(* CODESYS project ApplicationBase.library
   Author: FS
   Version: 1.0.8
   Description: All sample code provided by Beckhoff Automation LLC are for illustrative purposes only and are provided “as is” and without any warranties, express or implied. Actual implementations in applications will vary significantly. Beckhoff Automation LLC shall have no liability for, and does not waive any rights in relation to, any code samples that it provides or the use of such code samples for any purpose.
   Title: ApplicationBase
   DefaultNamespace: ApplicationBase
   Placeholder: ApplicationBase
   Company: Beckhoff Automation LLC

Project tree, tasks and I/O mapping:
  libraries: Tc2_DataExchange, 3.4.2.0 (Beckhoff Automation GmbH); Tc2_EtherCAT, 3.7.1.0 (Beckhoff Automation GmbH); Tc2_IoFunctions, 3.4.5.0 (Beckhoff Automation GmbH); Tc2_Math, 3.5.1.0 (Beckhoff Automation GmbH); Tc2_MC2, 3.3.72.0 (Beckhoff Automation GmbH); Tc2_MC2_Drive, 3.3.54.0 (Beckhoff Automation GmbH); Tc2_NcKinematicTransformation, 3.2.11.0 (Beckhoff Automation GmbH); Tc2_SerialCom, 3.4.6.0 (Beckhoff Automation GmbH); Tc2_Standard, 3.4.5.0 (Beckhoff Automation GmbH); Tc2_System, 3.10.1.0 (Beckhoff Automation GmbH); Tc2_TcpIp, 3.4.4.0 (Beckhoff Automation GmbH); Tc2_Utilities, 3.10.1.0 (Beckhoff Automation GmbH); Tc3_DynamicMemory, 1.1.4.0 (Beckhoff Automation GmbH); Tc3_EventLogger, 3.3.13.0 (Beckhoff Automation GmbH); Tc3_JsonXml, 3.4.7.0 (Beckhoff Automation GmbH); Tc3_Module, 3.4.5.0 (Beckhoff Automation GmbH); Tc3_PackML_V3, 1.0.6.0 (Beckhoff Automation GmbH)
  _Interface/
    interface I_Base
    interface I_Command: Execute
    interface I_Disposable: Dispose
    interface I_Enablable: Disable, Enable, Enabled
    interface I_Initializable: Initialize, Initialized
    interface I_Override: Override
    interface I_Resettable: Reset
    interface I_Simulatable: Simulated
    interface I_Stoppable: Stop, Stopped
    interface I_TaskResult: Busy, Error, ErrorId
    interface I_ToString: ToString
  _Internal/
    Collection/
      Interface/
        interface I_Collection: AddItem, Clear, Count, IsEmpty, RemoveItem
        interface I_Enumerator: Current, CurrentItem, MoveToNext, ResetIterator
      function block Collection [ST]: FillGaps, AddItem, Clear, Count, Current, CurrentItem, IsEmpty, MoveToNext, RemoveItem, ResetIterator
    CollectionPeeker/
      Interface/
        interface I_CollectionPeeker: CollectionName, FirstItem, LastItem, MoveDownOne, MoveUpOne, PageDown, PageUp, PeekAt, Refresh
        interface I_Peekable: AcceptPeeker
        interface I_Peeker: PeekCollection
      function block CollectionPeeker [ST]: RefreshItems, UpdateEndItem, UpdateFirstItem, CollectionName, FirstItem, Items, LastItem, MoveDownOne, MoveUpOne, PageDown, PageUp, PeekAt, PeekCollection, Refresh
    Component/
      Interface/
        interface I_ComponentCollection: Accept, Count, GetAtIndex, GetComponentByName
        interface I_ContainComponents: Components, DeregisterComponent, DeregisterCyclic, DeregisterInitialize, RegisterComponent, RegisterCyclic, RegisterInitialize
      function block ComponentCollection [ST]: Accept, AddComponent, Count, GetAtIndex, GetComponentByName, RemoveComponent
    Cyclic/
      Interface/
        interface I_Cyclic: CyclicLogic
      function block CyclicRunner [ST]: AddCallee, CallAll, RemoveCallee
    Events/
      function block TcEventClassArguments [ST]: AddString, Clear, Event
    Initialize/
      function block Initializer [ST]: AddInitialize, Initialized, Initializing, RemoveInitialize
    List/
      Interface/
        interface I_List: ContainsItem, GetAtIndex, InsertAtIndex, RemoveAtIndex
      function block List [ST]: AddItem, Clear, RemoveItem, CountListItems, ContainsItem, Count, GetAtIndex, InsertAtIndex, RemoveAtIndex
    Module/
      Interface/
        interface I_ContainModules: DeregisterCyclic, DeregisterInitialize, DeregisterModule, Modules, RegisterCyclic, RegisterInitialize, RegisterModule
        interface I_ModuleCollection: Accept, Count, GetAtIndex, GetModuleByName
      function block ModuleCollection [ST]: Accept, AddModule, Count, GetAtIndex, GetModuleByName, RemoveModule
    MotionTasks/
      AX5000/
        DUT/
          P_0_0074/
            data type ST_IDN_P_0_0074
            data type ST_IDN_P_0_0074_UDINT
          P_0_0074_LREAL/
            data type ST_IDN_P_0_0074_LREAL
          data type ST_AX5000AmpToNm
        function block MotionTask_AX5000AmpToNm [ST]: ActCurrent, ActTorque, Busy, CyclicLogic, Error, ErrorId, Execute
      Base/
        DUT/
          data type ST_TaskState
        function block MotionTask [ST]: Axis, Busy, CyclicLogic, Error, ErrorId, Execute, Name
        function block MotionTaskCollection [ST]: Busy, Error, ErrorId, ErrorTask, AddTask, CyclicLogic, FB_Init, RemoveTaskByInstance, Reset
      Coupling/
        function block MotionCoupleTask_Gearing [ST]: BufferMode, Busy, CyclicLogic, Error, ErrorId, Execute, GearIn, GearInMultiMasterOptions, GearRatioMaster1, GearRatioMaster2, GearRatioMaster3, GearRatioMaster4, Master1, Master2, Master3, Master4
      Home/
        function block MotionHomeTask_CoESetEncoderOffset [ST]: Busy, CyclicLogic, Error, ErrorId, Execute, HomePosition
        function block MotionHomeTask_SetPosition [ST]: Busy, CyclicLogic, Error, ErrorId, Execute, HomePosition
        function block MotionHomeTask_SetPositionOffset [ST]: Busy, CyclicLogic, Error, ErrorId, Execute, Feedback, HomePosition, Memory
        function block MotionHomeTask_SetZeroHere [ST]: Busy, CyclicLogic, Error, ErrorId, Execute
      Interface/
        interface I_AxisRef: Axis
        interface I_MotionJogTask: JogBackwards, JogForward, Mode, Position
        interface I_MotionPowerTask
        interface I_MotionTask: Axis, Name
        interface I_MotionTaskCollection: AddTask, ErrorTask, RemoveTaskByInstance
      Move/
        function block MoveAbsoluteTask [ST]: BufferMode, Busy, CyclicLogic, Error, ErrorId, Execute, MoveOptions, TargetPosition
        function block MoveJogTask [ST]: Busy, CyclicLogic, Error, ErrorId, Execute, JogBackwards, JogForward, Mode, Position
        function block MoveModuloTask [ST]: BufferMode, Busy, CyclicLogic, Direction, Error, ErrorId, Execute, MoveOptions, TargetPosition
        function block MoveRelativeTask [ST]: BufferMode, Busy, CyclicLogic, Error, ErrorId, Execute, MoveOptions, TargetDistance
        function block MoveVelocityTask [ST]: BufferMode, Busy, CyclicLogic, Error, ErrorId, Execute, MoveOptions, TargetVelocity
      Power/
        function block PowerTask [ST]: Busy, CyclicLogic, Disable, Enable, Enabled, Error, ErrorId, Execute, InhibitFeedBackward, InhibitFeedForward, Override
        function block StopTask [ST]: BufferMode, Busy, CyclicLogic, Error, ErrorId, Execute, MoveOptions
      Reset/
        function block CoEExtendedResetTask [ST]: Busy, CyclicLogic, Error, ErrorId, Execute
        function block CoEResetTask [ST]: Busy, CyclicLogic, Error, ErrorId, Execute
        function block SoEResetTask [ST]: Busy, CyclicLogic, Error, ErrorId, Execute
    Null/
      function block NullComponent [ST]
      function block NullItem [ST]
      function block NullModule [ST]: Accept, Components, DeregisterComponent, DeregisterCyclic, DeregisterInitialize, DeregisterModule, DeregisterWithParent, FB_Init, Modules, Name, RegisterComponent, RegisterCyclic, RegisterInitialize, RegisterModule, RegisterWithParent, ResetComponents, ResetModules
    Statemachine/
      Interface/
        interface I_StateList: AddStateAtIndex, GetStateAtIndex, NumberOfStates
      function block StateList [ST]: AddStateAtIndex, GetStateAtIndex, NumberOfStates
    Tracing/
      Interface/
        interface I_ContainTraceArgument: Arguments
        interface I_ContainTracePublisher: Publisher
        interface I_TraceArgument
        interface I_TraceInstanceLogger: LogMessageInstance
        interface I_TraceLogger: LogMessage
        interface I_TraceMessageInfo: Message, MessageId, Severity
        interface I_TracePublisher: Subscribe, Unsubscribe
        interface I_TraceSourceInfo: SourceId, SourceName, TimeStamp
      function block AdsLogger [ST]: FB_Init, LogMessage
      function block LocalLogger [ST]: ClearLog, LogMessage, Messages
      function block TcEventLogger [ST]: FB_Init, LogMessage
      function block TraceMessageInfo [ST]: Message, MessageId, Severity
      function block TraceSourceInfo [ST]: SourceId, SourceName, TimeStamp
      function USINT_To_TcEventSeverity [ST]
    Types/
      data type RegistrationResult
  Component/
    Interface/
      interface I_Component: Accept, DeregisterWithParent, Name, RegisterWithParent
      interface I_ComponentVisitor: VisitComponent
    function block Component [ST]: Accept, DeregisterWithParent, Name, RegisterWithParent, FB_Init
    function block CyclicComponent [ST]: CyclicLogic, DeregisterWithParent, RegisterWithParent
  Components/
    ADS/
      Interface/
        interface I_AdsAccess: AdsRW
        interface I_AdsRW: AmsNetId, AmsPort, Read, ReadBySymbol, Write, WriteBySymbol
      function block AdsReadWrite [ST]: Busy, Error, ErrorId, AdsComMode, AmsNetId, AmsPort, CyclicLogic, Read, ReadBySymbol, Write, WriteBySymbol
    Analog/
      DUT/
        data type ST_AnalogInputStatus_EL30xx
        data type ST_AnalogInputStatus_Generic
      Interface/
        interface I_AnalogChannel_Generic: DataValid, Error, Overrange, Underrange
        interface I_AnalogChannel_Standard: Limit1High, Limit1Low, Limit2High, Limit2Low
        interface I_AnalogInput: RawValue, Value
        interface I_AnalogOutput: RawValue, Value
      function block AnalogInput [ST]: CalibrateCustom, CalibrateLinear, FB_Init, Force, ForceValue, RawValue, Scale, Value
      function block AnalogInput_Generic [ST]: DataValid, Error, FB_Init, Overrange, Underrange
      function block AnalogInput_Standard [ST]: DataValid, Error, FB_Init, Limit1High, Limit1Low, Limit2High, Limit2Low, Overrange, Underrange
      function block AnalogOutput [ST]: CalibrateCustom, CalibrateLinear, FB_Init, Force, ForceValue, RawValue, Scale, Value
    CoE/
      DUT/
        data type ST_TerminalProductInfo
      Interface/
        interface I_CoeAccess: CoE
        interface I_CoeDevice: AdsAddr, Read, Write
      function block CoeDevice [ST]: Busy, Error, ErrorId, AdsAddr, CyclicLogic, Read, Write
      function block NullCoeDevice [ST]: AdsAddr, Busy, CyclicLogic, Error, ErrorId, Read, Write
    Cylinder/
      DUT/
        data type E_CylinderErrorId
        data type E_CylinderState
        data type ST_Cylinder_HMI
      Interface/
        interface I_Cylinder: ExtendTimeout, RetractTimeout
        interface I_CylinderCommand: Extend, Retract
        interface I_CylinderStatus: Extended, Extending, Retracted, Retracting
      function block Cylinder [ST]: CyclicLogic, Busy, Error, ErrorId, Extend, Extended, Extending, ExtendTimeout, Retract, Retracted, Retracting, RetractTimeout, Reset, FB_Init
      function block Cylinder_HMI [ST]: ExtendPermissive, RetractPermissive, ControlObject, CyclicLogic, ExtendCommandName, ExtendedName, FB_Init, RetractCommandName, RetractedName
      function block Cylinder_TcEvents [ST]: GetHighestActiveEventReaction, GetHighestActiveEventSeverity, Reset, SetEventReactions, CyclicLogic, FB_Init
    Digital/
      DUT/
        data type ST_DigitalInput_HMI
        data type ST_DigitalOutput_HMI
      Interface/
        interface I_DigitalInput: IsActive
        interface I_DigitalOutput: On
      Visitor/
        function block ForceVisitor [ST]: Force, VisitComponent
        function block ReleaseAllForceVisitor [ST]: ReleaseForces, VisitComponent, VisitModule
      function block DigitalInput_Combiner [ST]: AddInput, Force, IsActive
      function block DigitalInput_DebounceFallingEdge [ST]: CyclicLogic, DebounceTime, FB_Init, Force, IsActive
      function block DigitalInput_DebounceRisingEdge [ST]: CyclicLogic, DebounceTime, FB_Init, Force, IsActive
      function block DigitalInput_HMI [ST]: ControlObject, CyclicLogic, FB_Init
      function block DigitalInput_NC [ST]: FB_Init, Force, IsActive
      function block DigitalInput_NO [ST]: FB_Init, Force, IsActive
      function block DigitalOutput [ST]: FB_Init, Force, On
      function block DigitalOutput_HMI [ST]: ControlObject, CyclicLogic, FB_Init
    EtherCat/
      DUT/
        global variables EtherCatParameter
        data type ST_EtherCatMasterInfo
        data type ST_EtherCatSyncUnitTaskInfo
      Interface/
        interface I_EcIoDevice: Bootstrap, Configuration, DeviceError, Disabled, Init, InitCmdError, InvalidVPRS, OP, PreOp, SafeOp, State
        interface I_EtherCatDiagnosticEventProvider: RaiseEtherCatDiagnosticEvent, RaiseSyncUnitEvent
        interface I_EtherCatMasterDiagnostic: ConfiguredSlaveCount, GetIoDeviceByAddr, GetIoDeviceByName, LocalAmsNetId, MasterAmsNetId, RegisterEventProvider, SlaveCount
        interface I_IoDevice: IoDataValid
        interface I_SyncUnitTask: IoDataValid, IsHotConnect, SlaveCount
      function block EtherCatIoDevice [ST]: Bootstrap, CoE, Configuration, DeviceError, Disabled, Init, InitCmdError, InvalidVPRS, IoDataValid, OP, PreOp, SafeOp, State, AmsNetId, CyclicLogic, SyncUnit
      function block EtherCatMaster [ST]: FramesWcStatesOk, LookupMasterState, LookupSlaveState, MasterState, SlaveState, ConfiguredSlaveCount, GetIoDeviceByAddr, GetIoDeviceByName, LocalAmsNetId, MasterAmsNetId, RegisterEventProvider, SlaveCount, Initialize, Initialized, Reset, Busy, Error, ErrorId, CyclicLogic, FB_Init, Simulated
      function block EtherCatMaster_TcEvents [ST]: GetHighestActiveEventReaction, GetHighestActiveEventSeverity, RaiseEtherCatDiagnosticEvent, RaiseSyncUnitEvent, Reset, SetEventReactions, FB_Init
      function block SyncUnitTask [ST]: Initialize, Initialized, IoDataValid, IsHotConnect, IsTerminalPartOfSyncUnit, SlaveCount, Busy, Error, ErrorId, CyclicLogic, EventProvider, FB_Init, Simulated
    Recipe/
      Interface/
        interface I_RecipeManagment: AutoLoadChangesToActive, ChangesPending, LoadChangesToActive
      function block RecipeManagment [ST]: CyclicLogic, CompareData, AutoLoadChangesToActive, ChangesPending, LoadChangesToActive, FB_Init
    Safety/
      DUT/
        data type E_SafetyConnection_State
        data type E_SafetyEdm_State
        data type E_SafetyEStop_State
        data type E_SafetyGroup_Diag
        data type E_SafetyGroup_State
        data type E_SafetyMon_State
        data type E_SafetyOrAnd_State
        data type ST_SafetyAddressInfo
        data type ST_SafetyDeviceInfo
        data type ST_SafetyStateDiag
      Interface/
        interface I_InSafetyGroup: SafetyGroup
        interface I_SafetyBase: OK, ResetFunction
        interface I_SafetyModule: AddSafetyComponent, OK, SafetyPlcCoE
        interface I_SafetyReset: Execute, PulseDuration
        interface I_SafetySimulation: SimulateSafetyDiag, SimulateSafetyState
      Reset Function/
        function block SafetyResetPulse [ST]: CyclicLogic, Busy, Error, ErrorId, Execute, PulseDuration
      Visitor/
        function block SafetyOkVisitor [ST]: Check, OK, VisitComponent
        function block SetSafetySimulationVisitor [ST]: Diag, Simulated, State, VisitComponent
      function block SafetyAndOrFB [ST]: CyclicLogic
      function block SafetyBase [ST]: CyclicLogic, OK, Reset, ResetFunction, Simulated, SimulateSafetyDiag, SimulateSafetyState, Busy, Error, ErrorId
      function block SafetyConnectionFB_TcEvents [ST]: CyclicLogic, GetHighestActiveEventReaction, GetHighestActiveEventSeverity, Reset, SetEventReactions, FB_Init
      function block SafetyEdmFB_TcEvents [ST]: CyclicLogic, GetHighestActiveEventReaction, GetHighestActiveEventSeverity, Reset, SetEventReactions, FB_Init, SafetyGroup
      function block SafetyEstopFB_TcEvents [ST]: CyclicLogic, GetHighestActiveEventReaction, GetHighestActiveEventSeverity, Reset, SetEventReactions, ActiveName, FB_Init, SafetyGroup
      function block SafetyGroup_TcEvents [ST]: CyclicLogic, GetHighestActiveEventReaction, GetHighestActiveEventSeverity, Reset, SetEventReactions, AutoResetFaults, FB_Init
      function block SafetyModule [ST]: OnCyclicCall, Initializing, Simulated, SimulateSafetyDiag, SimulateSafetyState, Busy, Error, ErrorId, AddSafetyComponent, FB_Init, OK, Reset, SafetyAddressInfo, SafetyPlcCoE
      function block SafetyMonFB_TcEvents [ST]: CyclicLogic, GetHighestActiveEventReaction, GetHighestActiveEventSeverity, Reset, SetEventReactions, ActiveAlarm, ActiveName, FB_Init, SafetyGroup
    Serial/
      Interface/
        interface I_SerialByteConnection: ByteData, ByteDataRecieved, SendAByte
        interface I_SerialLineControl: rxBuffer, txBuffer
        interface I_SerialStringConnection: SendAString, StringData, StringRecieved
      function block SerialByteConnection [ST]: ByteData, ByteDataRecieved, CyclicLogic, FB_Init, Reset, SendAByte, SetDependencies
      function block SerialLineControl_ADS [ST]: CyclicLogic, rxBuffer, SetConnectionConfig, txBuffer
      function block SerialLineControl_Terminal [ST]: CyclicLogic, FB_Init, rxBuffer, SetConnectionConfig, SetDependencies, txBuffer
      function block SerialStringConnection [ST]: CyclicLogic, FB_Init, Reset, SendAString, SetDependencies, SetSerialConfiguration, StringData, StringRecieved
    Tcp Ip/
      DUT/
        data type ST_TcpIpPayload
      Interface/
        interface I_TcpIpConnection: ConnectionState, IP, Port, RegisterCommand, SendCommand, SendPriorityCommand, Socket
        interface I_TcpIpSubscription: UpdateCommandResult
      function block TcpIpCommandResultFilter [ST]: CyclicLogic, FB_Init, UpdateCommandResult
      function block TcpIpConnection [ST]: CyclicLogic, Initialize, Initialized, EvaluateResponse, GetNextCommand, GetNextPriorityCommand, SendReceiveSequence, ConnectionState, IP, PollTime, Port, ReceiveTimeout, ReconnectionTime, RegisterCommand, SendCommand, SendInterval, SendPriorityCommand, Socket
      global variables TcpIpConnectionParameter
  Events/
    Interface/
      interface I_EventArguments: AddString, Clear
      interface I_EventClass: Arguments, ClearEventById, IsResettable, RaiseEvent, ResetBySeverity, SetEvent
      interface I_EventClassTcEvents: GenerateTcEvents, GetHighestActiveEventSeverity
      interface I_EventReaction: GetHighestActiveEventReaction, SetEventReactions
      interface I_EventReactionTcEvents: GetHighestActiveEventSeverity
    function block TcEventClass [ST]: Dispose, FB_Exit, ClearEventById, GetHighestActiveEventReaction, GetHighestActiveEventSeverity, IsResettable, RaiseEvent, ResetBySeverity, SetEvent, SetEventReactions, CheckEventId, FindActiveSeverity, GetEventAutoResetInstance, GetEventInstance, GetEventTriggerInstance, SetEventTriggerInstance, Reset, Arguments, CyclicLogic, GenerateTcEvents
  HMI/
    DUT/
      data type ST_HmiFunction
    Interface/
      interface I_Button: Active, Name, Permissive
      interface I_HmiFunction: ControlType, Disable, Enable, Enabled, InstancePath, LinkObject
      interface I_Permissive: OK, Set
      interface I_StringCollection: AddString, Clear, Entries
    function block Button [ST]: Active, Name, Permissive
    function block HmiFunction [ST]: ControlObject, ControlType, CyclicLogic, Disable, Enable, Enabled, InstancePath, LinkObject
  Kinematic Group/
    Interface/
      interface I_KinematicGroup: AddAcsAxis, AddMcsAxis, BuildGroup, DissolveGroup, Status
    function block KinematicGroup [ST]: DeregisterWithParent, RegisterWithParent, CyclicLogic, Initialize, Initialized, AddAcsAxis, AddMcsAxis, BuildGroup, DissolveGroup, Override, Status, Reset, Busy, Error, ErrorId
    function block KinematicGroup_TcEvents [ST]: GetHighestActiveEventReaction, GetHighestActiveEventSeverity, Reset, SetEventReactions, CyclicLogic, FB_Init
  Modes/
    Interface/
      interface I_Mode: ChangeMode, CurrentMode
    function block ModeControl [ST]: ChangeMode, CurrentMode
    function block PackMLModeControl [ST]: ChangeMode, CurrentMode, CyclicLogic, StateMachine
  Module/
    Interface/
      interface I_Module: Accept, DeregisterWithParent, Name, RegisterWithParent, ResetComponents, ResetModules
      interface I_ModuleVisitor: VisitModule
    function block Module [ST]: FB_Init, CyclicLogic, OnCyclicCall, DeregisterComponent, DeregisterCyclic, DeregisterInitialize, DeregisterModule, DeregisterWithParent, Initialize, Initialized, Initializing, RegisterComponent, RegisterCyclic, RegisterInitialize, RegisterModule, RegisterWithParent, ResetComponents, ResetModules, Accept, Components, Modules, Name
  Module PackML/
    function block PackMLModule [ST]: FB_Init, Aborted, Aborting, Clearing, Completed, Completing, Execute, Held, Holding, Idle, Resetting, Starting, Stopped, Stopping, Suspended, Suspending, Unholding, Unsuspending, CyclicLogic, Statemachine, StateSelect
  Motion/
    DUT/
      data type ST_AxisPTP_HMI
      data type ST_MotionDefaults
    Interface/
      interface I_Axis: ErrorId, MotionTasks
      interface I_Axis_PTP
      interface I_AxisDynamics: Acceleration, BufferMode, Deceleration, Jerk, MoveOptions, Velocity
      interface I_AxisEnable: InhibitFeedBackward, InhibitFeedForward
      interface I_AxisGear: GearIn, GearInMultiMasterOptions, GearOut, GearRatioMaster1, GearRatioMaster2, GearRatioMaster3, GearRatioMaster4, Master1, Master2, Master3, Master4
      interface I_AxisHome: Home
      interface I_AxisJog: Jog
      interface I_AxisMoveAbsolute: MoveAbsolute
      interface I_AxisMoveModulo: MoveModulo
      interface I_AxisMoveRelative: MoveRelative
      interface I_AxisMoveVelocity: MoveVelocity
      interface I_AxisStatus: ActualAcceleration, ActualPosition, ActualPositionModulo, ActualTorque, ActualVelocity, AxisParameterSet, Enabled, PositionLag, SetAcceleration, SetPosition, SetPositionModulo, SetVelocity, Stopped
      interface I_SlaveAxis
    function block Axis [ST]: FB_Init, RegisterWithParent, CyclicLogic, Acceleration, BufferMode, Deceleration, Jerk, MoveOptions, Velocity, Disable, Enable, Enabled, InhibitFeedBackward, InhibitFeedForward, Override, Home, HomeTask, Initialize, Initialized, Jog, Reset, ResetTask, ActualAcceleration, ActualPosition, ActualPositionModulo, ActualTorque, ActualVelocity, AxisParameterSet, Busy, Error, ErrorId, PositionLag, SetAcceleration, SetPosition, SetPositionModulo, SetVelocity, Stop, Stopped, StopTask, Axis, MotionTasks
    function block Axis_TcEvents [ST]: GetHighestActiveEventReaction, GetHighestActiveEventSeverity, Reset, SetEventReactions, CyclicLogic, FB_Init
    function block AxisPTP [ST]: FB_Init, MoveAbsolute, MoveModulo, MoveRelative, MoveVelocity
    function block AxisPTP_HMI [ST]: DisablePermissive, EnablePermissive, HomePermissive, JogBackwardFastPermissive, JogBackwardSlowPermissive, JogForwardFastPermissive, JogForwardSlowPermissive, MoveAbsolutePermissive, MoveModuloPermissive, MoveRelativePermissive, MoveVelocityPermissive, ResetPermissive, StopPermissive, ControlObject, CyclicLogic, FB_Init
    function block SlaveAxisPTP [ST]: FB_Init, GearIn, GearInMultiMasterOptions, GearOut, GearRatioMaster1, GearRatioMaster2, GearRatioMaster3, GearRatioMaster4, Master1, Master2, Master3, Master4
  Permissive Interlock/
    function block PermissiveInterlock [ST]: Check, OK, Set
  Project Information/
    function F_GetCompany [ST]
    function F_GetTitle [ST]
    function F_GetVersion [ST]
  Statemachine/
    DUT/
      data type ST_PackMLStatemachine_HMI
      data type ST_Statemachine_HMI
    Generic/
      function NextMinorStep [ST]
      function NextStep [ST]
      function SetStep [ST]
      function block State [ST]: Executing, FB_Init, Inactive
      function block Statemachine [ST]: Mode, ChangeState, CurrentState, States, CyclicLogic
      function block Statemachine_HMI [ST]: ControlObject, CyclicLogic, FB_Init
    Interface/
      interface I_ContainStatemachine: Statemachine
      interface I_State: Executing, Inactive
      interface I_Statemachine: ChangeState, CurrentState, Mode, States
    PackML/
      function block NextAvailablePackMLCommands [ST]: GetCommands
      function block PackMLStatemachine [ST]: Mode, CallState, ChangeState, CurrentState, States, CyclicLogic
      function block PackMLStatemachine_HMI [ST]: ControlObject, CyclicLogic, FB_Init
      function block PackMLStatemachine_ModuleIntegrated [ST]: Mode, ChangeState, CurrentState, CyclicLogic, StateComplete, States
  Tracing/
    DUT/
      data type TcEventSeverityExt
    Interface/
      interface I_Trace: Critical, Error, Info, Verbose, Warning
    global variables CoreTrace
    function block Trace [ST]: Critical, Error, Info, LogMessage, Subscribe, TraceLevel, Unsubscribe, Verbose, Warning
  Utilities/
    AnyBuffer/
      DUT/
        data type ST_BufferConfiguration
        data type ST_BufferMetadata
      Interface/
        interface I_AnyBuffer: Clear, Configuration, DeleteAtIndex, isEmpty, isFull, Metadata, PeekAtIndex, PopAtIndex, PopLeft, PopRight, PushAtIndex, PushLeft, PushRight, ReplaceAtIndex
        interface I_AnyBufferStrategy: Clear, isEmpty, isFull
      TypedBuffers/
        function block FifoBuffer [ST]: Clear, FB_Init, isEmpty, isFull, Pop, Push
        function block LifoBuffer [ST]: Clear, FB_Init, isEmpty, isFull, Pop, Push
        function block ListBuffer [ST]: Clear, FB_Init, isEmpty, isFull, Pop, Push, removeOldest
        function block RingBuffer [ST]: AdvanceHead, AdvanceTail, Clear, FB_Init, isEmpty, isFull, Pop, Push
      function block AnyBuffer [ST]: buffer, Clear, Configuration, CountDecrement, CountIncrement, DeleteAtIndex, FB_Exit, FB_Init, FB_Reinit, isEmpty, isFull, Metadata, PeekAtIndex, PopAtIndex, PopLeft, PopRight, PushAtIndex, PushLeft, PushRight, ReplaceAtIndex
    File/
      DUT/
        data type ST_File_HMI
      Interface/
        interface I_FileHandler: ClearDocument, Datatype, LoadFile, nData, Path, pData, ReadSymbol, SaveFile, SymbolName, Timeout, UpdateSymbol
      function block File_HMI [ST]: LoadPermissive, SavePermissive, ControlObject, CyclicLogic, FB_Init
      function block JsonFile [ST]: CyclicLogic, ClearDocument, Datatype, LoadFile, nData, Path, pData, ReadSymbol, SaveFile, SymbolName, Timeout, UpdateSymbol, LoadFileSequence, SaveFileSequence, Reset, Busy, Error, ErrorId
      function block StringHelper [ST]: GetExtensionOrVarName, GetFileNameFromPath, GetFilePath, GetName, GetPath, GetSymbolPath, RemoveFirstChar, RemoveLastChar, StringToCharArray, ValidInput
    Flash/
      function block SyncedSquareWaves [ST]: Initialize, Initialized, CyclicLogic, Wave_0_5Hz, Wave_100Hz, Wave_1Hz, Wave_2Hz, Wave_500Hz, Wave_50Hz, Wave_5Hz
    Force/
      DUT/
        data type E_ForceState
      Interface/
        interface I_ForcibleBool: Force
        interface I_ForcibleInt: Force, ForceValue
      function block ForcibleBool [ST]: ResolveOutput, CurrentForceState, FB_Init, Input, Output, SetForceState
      function block ForcibleInt [ST]: ResolveOutput, CurrentForceState, FB_Init, ForceValue, Input, Output, SetForceState
    Functions/
      function CompareLREAL [ST]
      function CompareModulo [ST]
      function PercentToAnalog [ST]
    Scaling/
      Interface/
        interface I_AnalogScalable: Scale
        interface I_AnalogScale: InputMaximum, InputMinimum, OutputMaximum, OutputMinimum
        interface I_CalibratableLinear: CalibrateLinear
        interface I_CalibrateLinear: Gain, Offset
        interface I_TransformLRealValue: Transform
      function block AnalogScale [ST]: InputMaximum, InputMinimum, OutputMaximum, OutputMinimum, Transform
      function block Calibrate [ST]: Gain, Offset, Transform
    Timing/
      function block Stopwatch [ST]: Elapsed, Lap, Running, Start, Stop
  Version/
    global variables Global_Version
  Visitors/
    Enable/
      function block CheckComponentsEnabledVisitor [ST]: Check, Enabled, VisitComponent
      function block DisableAllComponentsVisitor [ST]: Disable, Enabled, VisitComponent
      function block EnableAllComponentsVisitor [ST]: Enable, Enabled, VisitComponent
    Events/
      function block GetActiveEventSeverityVisitor [ST]: ActiveEventSeverity, FB_Init, VisitComponent, VisitModule
    HMI/
      function block GetSystemTreeJsonHmiVisitor [ST]: Clear, FB_Init, GetTree, VisitComponent, VisitModule
      function block HmiEnableDisableAllVisitor [ST]: DisableHmi, EnableHmi, VisitComponent, VisitModule
    Override/
      function block SetAllOverrideVisitor [ST]: Set, VisitComponent, VisitModule
    PackML Statemachine/
      function block ChangePackMLStateOnAllSubModulesVisitor [ST]: ChangeState, VisitModule
      function block EventReactorPackMLVisitor [ST]: CyclicLogic, FB_Init, VisitComponent, VisitModule
    Reset/
      function block GetComponentsTaskResultVisitor [ST]: Busy, Error, ErrorId, Update, VisitComponent
      function block ResetAllVisitor [ST]: Busy, Error, ErrorId, Reset, VisitComponent, VisitModule
      function block ResetComponentsVisitor [ST]: Busy, Error, ErrorId, Reset, VisitComponent
      function block ResetModulesVisitor [ST]: Busy, Error, ErrorId, Reset, VisitModule
    Statemachine/
      function block ChangeModeOnAllSubModulesVisitor [ST]: ChangeMode, VisitModule
      function block ChangeStateOnAllSubModulesVisitor [ST]: ChangeState, VisitModule
      function block EventReactorVisitor [ST]: CyclicLogic, FB_Init, VisitComponent, VisitModule
    Stop/
      function block StopAllComponentsVisitor [ST]: Stop, Stopped, VisitComponent
  global variables ApplicationBaseMotionParameterNc2
  global variables ApplicationBaseParameter
*)

// _Internal/MotionTasks/AX5000/DUT/P_0_0074/ST_IDN_P_0_0074
TYPE ST_IDN_P_0_0074 :
	STRUCT
		Iq : ARRAY[0..9] OF UDINT; // Amps ( units := A x 100 )
		M  : ARRAY[0..9] OF UDINT; // Newton Meters ( units := Nm x 100 )
	END_STRUCT
END_TYPE

// _Internal/MotionTasks/AX5000/DUT/P_0_0074/ST_IDN_P_0_0074_UDINT
TYPE ST_IDN_P_0_0074_UDINT :
	STRUCT
		Actual	 : UINT;
		_Max	 : UINT;
		Elements : ST_IDN_P_0_0074;
	END_STRUCT
END_TYPE

// _Internal/MotionTasks/AX5000/DUT/P_0_0074_LREAL/ST_IDN_P_0_0074_LREAL
TYPE ST_IDN_P_0_0074_LREAL :
	STRUCT
		Iq : ARRAY[0..9] OF LREAL;
		M  : ARRAY[0..9] OF LREAL;
	END_STRUCT
END_TYPE

// _Internal/MotionTasks/AX5000/DUT/ST_AX5000AmpToNm
TYPE ST_AX5000AmpToNm :
	STRUCT
		Curve	   : ST_IDN_P_0_0074_LREAL; // Contents read in from P-0-0074   ( scaled )
		ActCurrent : LREAL;					// Actual current in Amps           ( units := A )
		ActTorque  : LREAL;					// Actual torque in Newton Meters   ( units := Nm )
	END_STRUCT
END_TYPE

// _Internal/MotionTasks/Base/DUT/ST_TaskState
TYPE ST_TaskState :
	STRUCT
		Name	: T_MaxString;
		Busy	: BOOL;
		Error	: BOOL;
		ErrorId : UDINT;
	END_STRUCT
END_TYPE

// _Internal/Types/RegistrationResult
{attribute 'qualified_only'}
{attribute 'strict'}
{attribute 'to_string'}
TYPE RegistrationResult :
(
	Succeeded := 0,
	NullReference := -1,
	TooManyComponents := -2,
	AlreadyAdded := -3,
	CollectionEmpty := -4,
	NotFoundInCollection := -5
);
END_TYPE

// Components/Analog/DUT/ST_AnalogInputStatus_EL30xx
{attribute 'pack_mode' := '1'}
TYPE ST_AnalogInputStatus_EL30xx :
	STRUCT
		Underrrange : BIT;
		Overrange	: BIT;
		Limit1L		: BIT;
		Limit1H		: BIT;
		Limit2L		: BIT;
		Limit2H		: BIT;
		Error		: BIT;
		TxPDOState	: BIT;
		TxPDOToggle : BIT;
	END_STRUCT
END_TYPE

// Components/Analog/DUT/ST_AnalogInputStatus_Generic
{attribute 'pack_mode' := '1'}
TYPE ST_AnalogInputStatus_Generic :
	STRUCT
		Underrrange : BIT;
		Overrange	: BIT;
		Error		: BIT;
		WcState		: BIT;
	END_STRUCT
END_TYPE

// Components/CoE/DUT/ST_TerminalProductInfo
{attribute 'pack_mode' := '2'}
TYPE ST_TerminalProductInfo : // Parameter 16#1018:0
	STRUCT
		Identity	 : WORD;
		VendorId	 : DINT;
		ProductCode	 : DINT;
		Revision	 : DINT;
		SerialNumber : DINT;
	END_STRUCT
END_TYPE

// Components/Cylinder/DUT/E_CylinderErrorId
{attribute 'qualified_only'}
TYPE E_CylinderErrorId : (
		NoError				  := 0,
		ExtendTimeout		  := 1,
		RetractTimeout		  := 2,
		ExtendedPlausibility  := 3,
		RetractedPlausibility := 4,
		BothSensorsActive	  := 5
	) UDINT;
END_TYPE

// Components/Cylinder/DUT/E_CylinderState
{attribute 'qualified_only'}
TYPE E_CylinderState : (
		Undefined  := 0,
		Extending  := 1,
		Extended   := 2,
		Retracting := 3,
		Retracted  := 4
	);
END_TYPE

// Components/Cylinder/DUT/ST_Cylinder_HMI
TYPE ST_Cylinder_HMI EXTENDS ST_HmiFunction :
	STRUCT
		Busy		  : BOOL;
		Error		  : BOOL;
		ErrorId		  : UDINT;
		Extended	  : BOOL;
		ExtendedName  : STRING := 'Extended';
		Retracted	  : BOOL;
		RetractedName : STRING := 'Retracted';
		Extend		  : Button;
		Retract		  : Button;
	END_STRUCT
END_TYPE

// Components/Digital/DUT/ST_DigitalInput_HMI
TYPE ST_DigitalInput_HMI EXTENDS ST_HmiFunction :
	STRUCT
		Active : BOOL;
		Force  : E_ForceState;
	END_STRUCT
END_TYPE

// Components/Digital/DUT/ST_DigitalOutput_HMI
TYPE ST_DigitalOutput_HMI EXTENDS ST_HmiFunction :
	STRUCT
		On	  : BOOL;
		Force : E_ForceState;
	END_STRUCT
END_TYPE

// Components/EtherCat/DUT/ST_EtherCatMasterInfo
TYPE ST_EtherCatMasterInfo :
	STRUCT
		AmsNetID	  : AMSNETID;
		DevID		  : UINT;
		DevState	  : UINT;
		ChangeCount	  : UINT;
		SlaveCount	  : UINT;
		CfgSlaveCount : UINT;
	END_STRUCT
END_TYPE

// Components/EtherCat/DUT/ST_EtherCatSyncUnitTaskInfo
TYPE ST_EtherCatSyncUnitTaskInfo :
	STRUCT
		WcState	   : BIT;
		ObjectId   : OTCID;
		State	   : UINT;
		SlaveCount : UINT;
	END_STRUCT
END_TYPE

// Components/Safety/DUT/E_SafetyConnection_State
{attribute 'qualified_only'}
{attribute 'strict'}
TYPE E_SafetyConnection_State : (
		Reset	   := 100,
		Session	   := 101,
		Connection := 102,
		Parameter  := 103,
		Data	   := 104,
		Shutdown   := 105,
		Deactive   := 106
	) USINT;
END_TYPE

// Components/Safety/DUT/E_SafetyEdm_State
{attribute 'qualified_only'}
TYPE E_SafetyEdm_State : (
		Invalid := 0,
		Stop	:= 2,
		Error	:= 4,
		Reset	:= 5,
		MonOff	:= 14,
		MonOn	:= 15
	) USINT;
END_TYPE

// Components/Safety/DUT/E_SafetyEStop_State
{attribute 'qualified_only'}
TYPE E_SafetyEStop_State : (
		Invalid	 := 0,
		Run		 := 1,
		Stop	 := 2,
		Safe	 := 3,
		Error	 := 4,
		Reset	 := 5,
		Start	 := 6,
		DelayOut := 7
	) USINT;
END_TYPE

// Components/Safety/DUT/E_SafetyGroup_Diag
{attribute 'qualified_only'}
TYPE E_SafetyGroup_Diag : (
		NoError		  := 0,
		FbError		  := 1,
		ComError	  := 2,
		ModuleError	  := 3,
		CmpError	  := 4,
		DeactiveError := 5,
		RestartError  := 6
	) UINT;
END_TYPE

// Components/Safety/DUT/E_SafetyGroup_State
{attribute 'qualified_only'}
TYPE E_SafetyGroup_State : (
		Invalid		 := 0,
		Run			 := 1,
		Stop		 := 2,
		Error		 := 4,
		Reset		 := 5,
		Start		 := 6,
		StopError	 := 7,
		Deactive	 := 16,
		WaitComError := 17
	) USINT;
END_TYPE

// Components/Safety/DUT/E_SafetyMon_State
{attribute 'qualified_only'}
TYPE E_SafetyMon_State : (
		Invalid	   := 0,
		Run		   := 1,
		Stop	   := 2,
		Safe	   := 3,
		Error	   := 4,
		Reset	   := 5,
		Start	   := 6,
		ErrorDelay := 7,
		DelayOut   := 8,
		FuncTest   := 9
	) USINT;
END_TYPE

// Components/Safety/DUT/E_SafetyOrAnd_State
{attribute 'qualified_only'}
TYPE E_SafetyOrAnd_State : (
		Invalid := 0,
		Run		:= 1,
		Stop	:= 2,
		Safe	:= 3
	) USINT;
END_TYPE

// Components/Safety/DUT/ST_SafetyAddressInfo
{attribute 'pack_mode' := '2'}
TYPE ST_SafetyAddressInfo : // Parameter 16#F980:0
	STRUCT
		FSoEAddress		  : WORD;
		SerialNumber	  : DINT;
		ProjectCRC		  : WORD;
		DefaultProjectCRC : WORD;
	END_STRUCT
END_TYPE

// Components/Safety/DUT/ST_SafetyDeviceInfo
{attribute 'pack_mode' := '2'}
TYPE ST_SafetyDeviceInfo : // Parameter 16#F9C0:0
	STRUCT
		DeviceName			 : STRING;
		SoftwareVersion		 : STRING;
		BootloaderVersion	 : STRING;
		SoftwareChecksum	 : DINT;
		BootmanagerChecksum	 : DINT;
		BootloaderChecksum	 : DINT;
		TwinSAFELogicVersion : DINT;
	END_STRUCT
END_TYPE

// Components/Safety/DUT/ST_SafetyStateDiag
{attribute 'pack_mode' := '1'}
TYPE ST_SafetyStateDiag :
	STRUCT
		State : USINT;
		Diag  : UINT; // **NOT PRESENT ON AND/OR FBs ** For components with USINT as Diag connection, connect first 8 Bit of UINT Diag. Inherited FB is evaluating correct length.
	END_STRUCT
END_TYPE

// Components/Tcp Ip/DUT/ST_TcpIpPayload
TYPE ST_TcpIpPayload :
	STRUCT
		Size : UDINT;
		Data : ARRAY[0..(TcpIpConnectionParameter.PayloadSize - 1)] OF BYTE;
	END_STRUCT
END_TYPE

// HMI/DUT/ST_HmiFunction
TYPE ST_HmiFunction :
	STRUCT
		Name	   : STRING;
		HmiEnabled : BOOL := TRUE;
	END_STRUCT
END_TYPE

// Motion/DUT/ST_AxisPTP_HMI
TYPE ST_AxisPTP_HMI EXTENDS ST_HmiFunction :
	STRUCT
		Unit				 : STRING;
		Busy				 : BOOL;
		Error				 : BOOL;
		ErrorId				 : UDINT;
		ActualAcceleration	 : LREAL;
		ActualPosition		 : LREAL;
		ActualPositionModulo : LREAL;
		ActualTorque		 : LREAL;
		ActualVelocity		 : LREAL;
		Status				 : ST_AxisStatus;
		Enable				 : Button;
		Disable				 : Button;
		Stop				 : Button;
		JogForwardSlow		 : Button;
		JogBackwardSlow		 : Button;
		JogForwardFast		 : Button;
		JogBackwardFast		 : Button;
		Home				 : Button;
		Reset				 : Button;
		MoveAbsolute		 : Button;
		TargetPosition		 : LREAL;
		MoveVelocity		 : Button;
		TargetVelocity		 : LREAL;
		MoveRelative		 : Button;
		TargetDistance		 : LREAL;
		MoveModulo			 : Button;
	END_STRUCT
END_TYPE

// Motion/DUT/ST_MotionDefaults
TYPE ST_MotionDefaults :
	STRUCT
		DefaultResetTask : CoEResetTask				  := (Name := 'MC Reset (CoE)');
		DefaultHomeTask	 : MotionHomeTask_SetZeroHere := (Name := 'MC Home');
		DefaultStopTask	 : StopTask					  := (Name := 'MC Stop');
	END_STRUCT
END_TYPE

// Statemachine/DUT/ST_PackMLStatemachine_HMI
TYPE ST_PackMLStatemachine_HMI EXTENDS ST_HmiFunction :
	STRUCT
		// Simplified Control
		ResetPermissive : BOOL;
		ResetPressed	: BOOL;
		Resetted		: BOOL;
		StartPermissive : BOOL;
		StartPressed	: BOOL;
		Started			: BOOL;
		StopPermissive	: BOOL;
		StopPressed		: BOOL;
		Stopped			: BOOL;
		// Standard Control
		CurrentMode	 : DINT;
		ModeCommand	 : DINT;
		CurrentState : E_PMLState;
		StateCommand : E_PMLCommand;
		// Next Available Commands
		NextAvailableCommands : ARRAY[0..9] OF E_PMLCommand;
	END_STRUCT
END_TYPE

// Statemachine/DUT/ST_Statemachine_HMI
TYPE ST_Statemachine_HMI EXTENDS ST_HmiFunction :
	STRUCT
		CurrentState	   : DINT;
		CurrentMode		   : DINT;
		StateChangeCommand : DINT;
		ModeChangeCommand  : DINT;
	END_STRUCT
END_TYPE

// Tracing/DUT/TcEventSeverityExt
{attribute 'qualified_only'}
{attribute 'strict'}
{attribute 'to_string'}
TYPE TcEventSeverityExt : (
		Verbose	 := 0,
		Info	 := 1,
		Warning	 := 2,
		Error	 := 3,
		Critical := 4,
		Off		 := 5
	);
END_TYPE

// Utilities/AnyBuffer/DUT/ST_BufferConfiguration
TYPE ST_BufferConfiguration :
	STRUCT
		isPersistent	 : BOOL; // is the buffer persistent?
		capacity		 : DINT; // No of elements in buffer
		elementSize		 : DINT; // Buffer element size in bytes
		bufferSize		 : DINT; // Complete buffer size in bytes	
		bufferBoundLower : DINT; // Lower boundary of the buffer
		bufferBoundUpper : DINT; // Upper boundary of the buffer	
	END_STRUCT
END_TYPE

// Utilities/AnyBuffer/DUT/ST_BufferMetadata
TYPE ST_BufferMetadata :
	STRUCT
		headIndex	 : DINT;
		tailIndex	 : DINT;
		capacity	 : DINT;
		elementCount : DINT;
	END_STRUCT
END_TYPE

// Utilities/File/DUT/ST_File_HMI
TYPE ST_File_HMI EXTENDS ST_HmiFunction :
	STRUCT
		Path	: STRING;
		Load	: Button;
		Save	: Button;
		NewPath : BOOL;
	END_STRUCT
END_TYPE

// Utilities/Force/DUT/E_ForceState
{attribute 'qualified_only'}
{attribute 'strict'}
{attribute 'to_string'}
TYPE E_ForceState : (
		Unforced := 0,
		ForceOn	 := 1,
		ForceOff := 2
	) DINT;
END_TYPE

// Components/EtherCat/DUT/EtherCatParameter
VAR_GLOBAL CONSTANT
	MAX_EC_SLAVES : UINT := 49;
END_VAR

// Components/Tcp Ip/TcpIpConnectionParameter
{attribute 'qualified_only'}
VAR_GLOBAL CONSTANT
	PayloadSize : UDINT := 1460; // Payload in Bytes
END_VAR

// Tracing/CoreTrace
VAR_GLOBAL
	Trace : Trace<ApplicationBaseParameter.MaxCountInCollections> := (TraceLevel := ApplicationBaseParameter.TraceLevel);
	{attribute 'hide'}
	TcEventLogger : TcEventLogger(Trace);
	{attribute 'hide'}
	AdsLogger : AdsLogger(Trace);
END_VAR

// Version/Global_Version
{attribute 'TcGenerated'}
{attribute 'no-analysis'}
{attribute 'linkalways'}
// This function has been automatically generated from the project information.
VAR_GLOBAL CONSTANT
	{attribute 'const_non_replaced'}
	stLibVersion_ApplicationBase : ST_LibVersion := (iMajor := 1, iMinor := 0, iBuild := 8, iRevision := 0, nFlags := 0, sVersion := '1.0.8');
END_VAR

// ApplicationBaseMotionParameterNc2
{attribute 'qualified_only'}
VAR_GLOBAL CONSTANT
	MaxMotionTasks : UDINT := 10;
END_VAR

// ApplicationBaseParameter
{attribute 'qualified_only'}
VAR_GLOBAL CONSTANT
	MaxCountInCollections : UDINT			   := 50;
	EnableTcEventLogging  : BOOL			   := FALSE;
	EnableAdsLogger		  : BOOL			   := TRUE;
	ClearingTimeout		  : TIME			   := T#2S;
	TraceLevel			  : TcEventSeverityExt := TcEventSeverityExt.Verbose;
END_VAR

// _Interface/I_Base
INTERFACE I_Base EXTENDS __SYSTEM.IQueryInterface

END_INTERFACE

// _Interface/I_Command
INTERFACE I_Command EXTENDS I_Base

METHOD Execute : BOOL
VAR_INPUT
END_VAR
END_METHOD

END_INTERFACE

// _Interface/I_Disposable
INTERFACE I_Disposable EXTENDS I_Base

METHOD Dispose
VAR_INPUT
END_VAR
END_METHOD

END_INTERFACE

// _Interface/I_Enablable
INTERFACE I_Enablable EXTENDS I_Base

METHOD Disable
VAR_INPUT
END_VAR
END_METHOD

METHOD Enable
VAR_INPUT
END_VAR
END_METHOD

{attribute 'monitoring' := 'call'}
PROPERTY Enabled : BOOL
GET
END_GET
END_PROPERTY

END_INTERFACE

// _Interface/I_Initializable
INTERFACE I_Initializable EXTENDS I_Base

METHOD Initialize
END_METHOD

{attribute 'monitoring' := 'call'}
PROPERTY Initialized : BOOL
GET
END_GET
SET
END_SET
END_PROPERTY

END_INTERFACE

// _Interface/I_Override
INTERFACE I_Override EXTENDS I_Base

{attribute 'monitoring' := 'call'}
PROPERTY Override : LREAL
SET
END_SET
END_PROPERTY

END_INTERFACE

// _Interface/I_Resettable
INTERFACE I_Resettable EXTENDS I_Base

METHOD Reset
END_METHOD

END_INTERFACE

// _Interface/I_Simulatable
INTERFACE I_Simulatable EXTENDS I_Base

{attribute 'monitoring' := 'call'}
PROPERTY Simulated : BOOL
GET
END_GET
SET
END_SET
END_PROPERTY

END_INTERFACE

// _Interface/I_Stoppable
INTERFACE I_Stoppable EXTENDS I_Base

METHOD Stop
VAR_INPUT
END_VAR
END_METHOD

{attribute 'monitoring' := 'call'}
PROPERTY Stopped : BOOL
GET
END_GET
END_PROPERTY

END_INTERFACE

// _Interface/I_TaskResult
INTERFACE I_TaskResult EXTENDS I_Base

{attribute 'monitoring' := 'call'}
PROPERTY Busy : BOOL
GET
END_GET
END_PROPERTY

{attribute 'monitoring' := 'call'}
PROPERTY Error : BOOL
GET
END_GET
END_PROPERTY

{attribute 'monitoring' := 'call'}
PROPERTY ErrorId : UDINT
GET
END_GET
END_PROPERTY

END_INTERFACE

// _Interface/I_ToString
INTERFACE I_ToString EXTENDS I_Base

METHOD ToString : T_MaxString
VAR_INPUT
END_VAR
END_METHOD

END_INTERFACE

// _Internal/Collection/Interface/I_Collection
INTERFACE I_Collection EXTENDS I_Enumerator

METHOD AddItem
VAR_INPUT
	Item : I_Base;
END_VAR
END_METHOD

METHOD Clear
VAR_INPUT
END_VAR
END_METHOD

{attribute 'monitoring' := 'call'}
PROPERTY Count : UDINT
GET
END_GET
END_PROPERTY

{attribute 'monitoring' := 'call'}
PROPERTY IsEmpty : BOOL
GET
END_GET
END_PROPERTY

METHOD RemoveItem
VAR_INPUT
	Item : I_Base;
END_VAR
END_METHOD

END_INTERFACE

// _Internal/Collection/Interface/I_Enumerator
INTERFACE I_Enumerator

PROPERTY Current : I_Base
GET
END_GET
END_PROPERTY

{attribute 'monitoring' := 'call'}
PROPERTY CurrentItem : UDINT
GET
END_GET
END_PROPERTY

PROPERTY MoveToNext : BOOL
GET
END_GET
END_PROPERTY

METHOD ResetIterator
VAR_INPUT
END_VAR
END_METHOD

END_INTERFACE

// _Internal/Collection/Collection
FUNCTION_BLOCK Collection
VAR_GENERIC CONSTANT
	CollectionSize : UDINT := 1;
END_VAR IMPLEMENTS I_Collection, I_Enumerator
VAR
	{attribute 'instance-path'}
	{attribute 'noinit'}
	InstancePath  : STRING;
	_Data		  : ARRAY[0..CollectionSize - 1] OF I_Base;
	_Current	  : I_Base;
	_Count		  : UDINT;
	_CurrentIndex : UDINT;
	{attribute 'hide'}
	NullItem : NullItem;
	{attribute 'hide'}
	ipNullItem : I_Base := NullItem;
END_VAR

METHOD PROTECTED FillGaps
VAR
	Item	 : I_Base;
	ItemNext : I_Base;
	i		 : UDINT;
END_VAR
IF _Count > 1 THEN
	FOR i := 0 TO (_Count - 2) DO
		Item	 := _Data[i];
		ItemNext := _Data[i + 1];
		IF Item = 0 AND ItemNext <> 0 THEN
			_Data[i]	 := ItemNext;
			_Data[i + 1] := 0;
		END_IF
	END_FOR
END_IF
END_METHOD

METHOD AddItem
VAR_INPUT
	Item	: I_Base;
END_VAR
IF Item = 0 THEN
	Trace.Error(InstancePath, 'No Items to add to this Collection!');
	RETURN;
END_IF

IF _Count >= CollectionSize - 1 THEN
	Trace.Error(InstancePath, 'No space left in Collection, increase size!');
	RETURN;
END_IF

_Data[_Count] := Item;
_Count		  := _Count + 1;
END_METHOD

METHOD Clear
VAR
	i : UDINT;
END_VAR
IF _Count = 0 THEN
	RETURN;
END_IF

FOR i := 0 TO _Count - 1 DO
	_Data[i] := 0;
END_FOR

_Count := 0;
ResetIterator();
END_METHOD

{attribute 'monitoring' := 'call'}
PROPERTY Count : UDINT
GET
Count := _Count;
END_GET
END_PROPERTY

PROPERTY Current : I_Base
GET
IF _Current <> 0 THEN
	Current := _Current; 
END_IF
END_GET
END_PROPERTY

{attribute 'monitoring' := 'call'}
PROPERTY CurrentItem : UDINT
GET
CurrentItem := _CurrentIndex;
END_GET
END_PROPERTY

{attribute 'monitoring' := 'call'}
PROPERTY IsEmpty : BOOL
GET
IsEmpty := _Count = 0;
END_GET
END_PROPERTY

PROPERTY MoveToNext : BOOL
GET
MoveToNext := FALSE;
IF Count = 0 THEN
	RETURN;
END_IF

IF _CurrentIndex = Count THEN
	RETURN;
END_IF

_Current	  := _Data[_CurrentIndex];
_CurrentIndex := _CurrentIndex + 1;
MoveToNext	  := TRUE;
END_GET
END_PROPERTY

METHOD RemoveItem
VAR_INPUT
	Item : I_Base;
END_VAR

VAR
	i		  : UDINT;
	ItemFound : BOOL;
END_VAR
IF _Count = 0 THEN
	Trace.LogMessage(InstancePath, 'No Items found in this Collection!');
	RETURN;
END_IF

IF Item = 0 THEN
	Trace.LogMessage(InstancePath, 'Item to remove needs to be valid interface!');
	RETURN;
END_IF

FOR i := 0 TO (_Count - 1) DO
	IF _Data[i] = Item THEN
		_Data[i]  := 0;
		ItemFound := TRUE;
	END_IF
END_FOR

FillGaps();
IF ItemFound THEN
	_Count := _Count - 1;
END_IF
END_METHOD

METHOD ResetIterator
_Current	  := ipNullItem;
_CurrentIndex := 0;
END_METHOD

END_FUNCTION_BLOCK

// _Internal/Null/NullItem
FUNCTION_BLOCK NullItem IMPLEMENTS I_Base
VAR
END_VAR

END_FUNCTION_BLOCK

// Tracing/Trace
FUNCTION_BLOCK Trace
VAR_GENERIC CONSTANT
	MaxCount : UDINT := 10;
END_VAR IMPLEMENTS I_TracePublisher, I_Trace, I_TraceLogger
VAR
	Loggers : ARRAY[0..MaxCount] OF I_TraceLogger;
	_TraceLevel : TcEventSeverityExt := TcEventSeverityExt.Warning;
END_VAR

METHOD Critical
VAR_INPUT
	Source	  : T_MaxString;
	Message	  : T_MaxString;
END_VAR
VAR
	i : UDINT;
END_VAR
FOR i := 0 TO MaxCount DO
	IF Loggers[i] <> 0 AND_THEN _TraceLevel < 5 THEN
		Loggers[i].LogMessage(Source,
							  Message,
							  0,
							  0,
							  1,
							  4);
	END_IF
END_FOR
END_METHOD

METHOD Error
VAR_INPUT
	Source	  : T_MaxString;
	Message	  : T_MaxString;
END_VAR
VAR
	i : UDINT;
END_VAR
FOR i := 0 TO MaxCount DO
	IF Loggers[i] <> 0 AND_THEN _TraceLevel < 4 THEN
		Loggers[i].LogMessage(Source,
							  Message,
							  0,
							  0,
							  1,
							  3);
	END_IF
END_FOR
END_METHOD

METHOD Info
VAR_INPUT
	Source	  : T_MaxString;
	Message	  : T_MaxString;
END_VAR
VAR
	i : UDINT;
END_VAR
FOR i := 0 TO MaxCount DO
	IF Loggers[i] <> 0 AND_THEN _TraceLevel < 2 THEN
		Loggers[i].LogMessage(Source,
							  Message,
							  0,
							  0,
							  1,
							  1);
	END_IF
END_FOR
END_METHOD

METHOD LogMessage
VAR_INPUT
	Key		  : T_MaxString;
	Value	  : T_MaxString;
	SourceId  : UDINT := 0;
	TimeStamp : ULINT := 0;
	MessageId : UDINT := 1;
	Severity  : USINT := 1;
END_VAR

VAR
	i : UDINT;
END_VAR
FOR i := 0 TO MaxCount DO
	IF Loggers[i] <> 0 THEN
		Loggers[i].LogMessage(Key,
							  Value,
							  SourceId,
							  TimeStamp,
							  MessageId,
							  Severity);
	END_IF
END_FOR
END_METHOD

METHOD Subscribe
VAR_INPUT
	Logger : I_TraceLogger;
END_VAR

VAR
	i : UDINT;
END_VAR
FOR i := 0 TO ApplicationBaseParameter.MaxCountInCollections DO
	IF Loggers[i] = 0 THEN
		Loggers[i] := Logger;
		EXIT;
	END_IF
END_FOR
END_METHOD

PROPERTY TraceLevel : TcEventSeverityExt
GET
TraceLevel := _TraceLevel;
END_GET
SET
_TraceLevel := TraceLevel;
END_SET
END_PROPERTY

METHOD Unsubscribe
VAR_INPUT
	Logger : I_TraceLogger;
END_VAR

VAR
	i : UDINT;
END_VAR
FOR i := 0 TO ApplicationBaseParameter.MaxCountInCollections DO
	IF Loggers[i] = Logger THEN
		Loggers[i] := 0;
		EXIT;
	END_IF
END_FOR
END_METHOD

METHOD Verbose
VAR_INPUT
	Source	  : T_MaxString;
	Message	  : T_MaxString;
END_VAR
VAR
	i : UDINT;
END_VAR
FOR i := 0 TO MaxCount DO
	IF Loggers[i] <> 0 AND_THEN _TraceLevel = 0 THEN
		Loggers[i].LogMessage(Source,
							  Message,
							  0,
							  0,
							  1,
							  0);
	END_IF
END_FOR
END_METHOD

METHOD Warning
VAR_INPUT
	Source	  : T_MaxString;
	Message	  : T_MaxString;
END_VAR
VAR
	i : UDINT;
END_VAR
FOR i := 0 TO MaxCount DO
	IF Loggers[i] <> 0 AND_THEN _TraceLevel < 3 THEN
		Loggers[i].LogMessage(Source,
							  Message,
							  0,
							  0,
							  1,
							  2);
	END_IF
END_FOR
END_METHOD

END_FUNCTION_BLOCK

// _Internal/Tracing/Interface/I_TracePublisher
INTERFACE I_TracePublisher

METHOD Subscribe
VAR_INPUT
	Logger : I_TraceLogger;
END_VAR
END_METHOD

METHOD Unsubscribe
VAR_INPUT
	Logger : I_TraceLogger;
END_VAR
END_METHOD

END_INTERFACE

// _Internal/Tracing/Interface/I_TraceLogger
INTERFACE I_TraceLogger EXTENDS I_Base

METHOD LogMessage
VAR_INPUT
	Key		  : T_MaxString;
	Value	  : T_MaxString;
	SourceId  : UDINT := 0;
	TimeStamp : ULINT := 0;
	MessageId : UDINT := 1;
	Severity  : USINT := 1;
END_VAR
END_METHOD

END_INTERFACE

// Tracing/Interface/I_Trace
INTERFACE I_Trace

METHOD Critical
VAR_INPUT
	Source	  : T_MaxString;
	Message	  : T_MaxString;
END_VAR
END_METHOD

METHOD Error
VAR_INPUT
	Source	  : T_MaxString;
	Message	  : T_MaxString;
END_VAR
END_METHOD

METHOD Info
VAR_INPUT
	Source	  : T_MaxString;
	Message	  : T_MaxString;
END_VAR
END_METHOD

METHOD Verbose
VAR_INPUT
	Source	  : T_MaxString;
	Message	  : T_MaxString;
END_VAR
END_METHOD

METHOD Warning
VAR_INPUT
	Source	  : T_MaxString;
	Message	  : T_MaxString;
END_VAR
END_METHOD

END_INTERFACE

// _Internal/CollectionPeeker/Interface/I_CollectionPeeker
INTERFACE I_CollectionPeeker EXTENDS I_Base

{attribute 'monitoring':='call'}
PROPERTY CollectionName : T_MaxString
GET
END_GET
SET
END_SET
END_PROPERTY

{attribute 'monitoring':='call'}
PROPERTY FirstItem : UDINT
GET
END_GET
END_PROPERTY

{attribute 'monitoring':='call'}
PROPERTY LastItem : UDINT
GET
END_GET
END_PROPERTY

{attribute 'monitoring' := 'call'}
PROPERTY MoveDownOne : BOOL
SET
END_SET
END_PROPERTY

{attribute 'monitoring' := 'call'}
PROPERTY MoveUpOne : BOOL
SET
END_SET
END_PROPERTY

{attribute 'monitoring' := 'call'}
PROPERTY PageDown : BOOL
SET
END_SET
END_PROPERTY

{attribute 'monitoring' := 'call'}
PROPERTY PageUp : BOOL
SET
END_SET
END_PROPERTY

METHOD PeekAt
VAR_INPUT
	Peekable : I_Peekable;
END_VAR
END_METHOD

{attribute 'monitoring':='call'}
PROPERTY Refresh : BOOL
GET
END_GET
SET
END_SET
END_PROPERTY

END_INTERFACE

// _Internal/CollectionPeeker/Interface/I_Peekable
INTERFACE I_Peekable EXTENDS I_Base

METHOD AcceptPeeker
VAR_INPUT
	Peeker : I_Peeker;
END_VAR
END_METHOD

END_INTERFACE

// _Internal/CollectionPeeker/Interface/I_Peeker
INTERFACE I_Peeker EXTENDS I_Base

METHOD PeekCollection
VAR_INPUT
	Collection : I_Collection;
END_VAR
END_METHOD

END_INTERFACE

// _Internal/CollectionPeeker/CollectionPeeker
{attribute 'hide_all_locals'}
FUNCTION_BLOCK CollectionPeeker
VAR_GENERIC CONSTANT
	Peek_Size : UDINT := 5;
END_VAR IMPLEMENTS I_CollectionPeeker, I_Peeker
VAR
	_CurrentItem	: UDINT;
	_EndItem		: UDINT;
	_CollectionName : T_MaxString;
	_Collection		: I_Collection;
	_Items			: ARRAY[1..Peek_Size] OF I_Base;
END_VAR

METHOD PRIVATE RefreshItems
VAR
	startItem  : UDINT;
	endItem	   : UDINT;
	i		   : UDINT := 1;
	wrapAround : BOOL;
END_VAR
MEMSET(ADR(_Items), 0, SIZEOF(_Items));
IF _CurrentItem > _EndItem THEN //we're wrapped around
	i		   := 1 + ((_Collection.Count - _CurrentItem) + 1);
	wrapAround := TRUE;
END_IF

_Collection.ResetIterator();
WHILE _Collection.MoveToNext DO
	IF _Collection.CurrentItem >= _CurrentItem AND _Collection.CurrentItem <= _EndItem THEN
		_Items[i] := _Collection.Current;
		i		  := i + 1;
	ELSIF wrapAround AND (_Collection.CurrentItem >= _CurrentItem OR _Collection.CurrentItem <= _EndItem) THEN
		_Items[i] := _Collection.Current;
		i		  := i + 1;
		IF i > Peek_Size THEN
			i := 1;
		END_IF
	END_IF
END_WHILE
END_METHOD

METHOD PRIVATE UpdateEndItem
VAR_INPUT
END_VAR
_EndItem := _CurrentItem + Peek_Size - 1;
IF _EndItem > _Collection.Count THEN
	_EndItem := _EndItem - _Collection.Count;
END_IF
END_METHOD

METHOD PRIVATE UpdateFirstItem
VAR_INPUT
END_VAR
END_METHOD

{attribute 'monitoring':='call'}
PROPERTY CollectionName : T_MaxString
GET
CollectionName := _CollectionName;
END_GET
SET
_CollectionName := CollectionName;
END_SET
END_PROPERTY

{attribute 'monitoring' := 'call'}
PROPERTY FirstItem : UDINT
GET
FirstItem := _CurrentItem;
END_GET
SET
IF _Collection = 0 THEN
	RETURN;
END_IF

IF FirstItem > _Collection.Count OR FirstItem < 1 THEN
	RETURN;
END_IF

_CurrentItem := FirstItem;
UpdateEndItem();
RefreshItems();
END_SET
END_PROPERTY

{attribute 'monitoring' := 'call'}
PROPERTY Items : REFERENCE TO ARRAY[1..Peek_Size] OF I_Base
GET
Items REF= _Items;
END_GET
END_PROPERTY

{attribute 'monitoring' := 'call'}
PROPERTY LastItem : UDINT
GET
LastItem := _EndItem;
END_GET
END_PROPERTY

{attribute 'monitoring' := 'call'}
PROPERTY MoveDownOne : BOOL
GET
END_GET
SET
IF _Collection = 0 OR NOT MoveDownOne THEN
	RETURN;
END_IF

IF _Collection.Count <= Peek_Size THEN
	RETURN;
END_IF

_CurrentItem := _CurrentItem + 1;
IF _CurrentItem > _Collection.Count THEN
	_CurrentItem := 1;
END_IF

UpdateEndItem();
RefreshItems();
END_SET
END_PROPERTY

{attribute 'monitoring' := 'call'}
PROPERTY MoveUpOne : BOOL
GET
END_GET
SET
IF _Collection = 0 THEN
	RETURN;
END_IF

IF _Collection.Count <= Peek_Size THEN
	RETURN;
END_IF

_CurrentItem := _CurrentItem - 1;
IF _CurrentItem < 1 THEN
	_CurrentItem := _Collection.Count;
END_IF

UpdateEndItem();
RefreshItems();
END_SET
END_PROPERTY

{attribute 'monitoring' := 'call'}
PROPERTY PageDown : BOOL
GET
END_GET
SET
IF _Collection = 0 OR NOT PageDown THEN
	RETURN;
END_IF

IF _Collection.Count <= Peek_Size THEN
	RETURN;
END_IF

IF _CurrentItem > (_Collection.Count - Peek_Size) THEN
	_CurrentItem := (Peek_Size - (_Collection.Count - _CurrentItem));
ELSE
	_CurrentItem := _CurrentItem + Peek_Size;
END_IF

UpdateEndItem();
RefreshItems();
END_SET
END_PROPERTY

{attribute 'monitoring' := 'call'}
PROPERTY PageUp : BOOL
GET
END_GET
SET
VAR
	tmp : UDINT;
END_VAR
IF _Collection = 0 OR NOT PageUp THEN
	RETURN;
END_IF

IF _Collection.Count <= Peek_Size THEN
	RETURN;
END_IF

IF _CurrentItem < Peek_Size THEN
	_CurrentItem := (_Collection.Count - (Peek_Size - _CurrentItem));
ELSE
	_CurrentItem := _CurrentItem - Peek_Size;
END_IF

UpdateEndItem();
RefreshItems();
END_SET
END_PROPERTY

METHOD PeekAt
VAR_INPUT
	Peekable : I_Peekable;
END_VAR
Peekable.AcceptPeeker(THIS^);
END_METHOD

METHOD PeekCollection
VAR_INPUT
	Collection : I_Collection;
END_VAR
_Collection	 := Collection;
_CurrentItem := 1;
_EndItem	 := Peek_Size;
RefreshItems();
END_METHOD

{attribute 'monitoring':='call'}
PROPERTY Refresh : BOOL
GET
END_GET
SET
IF _Collection <> 0 AND Refresh THEN
	RefreshItems();
END_IF
END_SET
END_PROPERTY

END_FUNCTION_BLOCK

// _Internal/Component/Interface/I_ComponentCollection
INTERFACE I_ComponentCollection EXTENDS I_Base

METHOD Accept
VAR_INPUT
	Visitor : I_ComponentVisitor;
END_VAR
END_METHOD

{attribute 'monitoring' := 'call'}
PROPERTY Count : UDINT
GET
END_GET
END_PROPERTY

METHOD GetAtIndex : I_Component
VAR_INPUT
	Index : UDINT;
END_VAR
END_METHOD

METHOD GetComponentByName : I_Component
VAR_INPUT
	Name : T_MaxString;
END_VAR
END_METHOD

END_INTERFACE

// Component/Interface/I_ComponentVisitor
INTERFACE I_ComponentVisitor

METHOD VisitComponent
VAR_INPUT
	Component : I_Component;
END_VAR
END_METHOD

END_INTERFACE

// Component/Component
FUNCTION_BLOCK ABSTRACT Component IMPLEMENTS I_Component
VAR
	_Name : T_MaxString;
	RegisteredAsComponentResult : RegistrationResult;
END_VAR

METHOD Accept
VAR_INPUT
	ComponentVisitor : I_ComponentVisitor;
END_VAR
ComponentVisitor.VisitComponent(THIS^);
END_METHOD

METHOD DeregisterWithParent
VAR_INPUT
	Parent : I_ContainComponents;
END_VAR
Parent.DeregisterComponent(THIS^);
END_METHOD

{attribute 'monitoring' := 'call'}
PROPERTY Name : T_MaxString
GET
Name := _Name;
END_GET
SET
_Name := Name;
END_SET
END_PROPERTY

METHOD RegisterWithParent
VAR_INPUT
	Parent : I_ContainComponents;
END_VAR
RegisteredAsComponentResult := Parent.RegisterComponent(THIS^);
END_METHOD

//FB_Init is always available implicitly and it is used primarily for initialization.

//The return value is not evaluated. For a specific influence, you can also declare the

//methods explicitly and provide additional code there with the standard initialization

//code. You can evaluate the return value.
METHOD FB_Init : BOOL
VAR_INPUT
	bInitRetains : BOOL; // TRUE: the retain variables are initialized (reset warm / reset cold)
	bInCopyCode	 : BOOL; // TRUE: the instance will be copied to the copy code afterward (online change)   
	Name		 : T_MaxString;
END_VAR
_Name := Name;
END_METHOD

END_FUNCTION_BLOCK

// Component/Interface/I_Component
INTERFACE I_Component EXTENDS I_Base

METHOD Accept
VAR_INPUT
	ComponentVisitor : I_ComponentVisitor;
END_VAR
END_METHOD

METHOD DeregisterWithParent
VAR_INPUT
	Parent : I_ContainComponents;
END_VAR
END_METHOD

{attribute 'monitoring' := 'call'}
PROPERTY Name : T_MaxString
GET
END_GET
SET
END_SET
END_PROPERTY

METHOD RegisterWithParent
VAR_INPUT
	Parent : I_ContainComponents;
END_VAR
END_METHOD

END_INTERFACE

// _Internal/Component/Interface/I_ContainComponents
INTERFACE I_ContainComponents EXTENDS I_Base

PROPERTY Components : I_ComponentCollection
GET
END_GET
END_PROPERTY

METHOD DeregisterComponent  : RegistrationResult
VAR_INPUT
	Component : I_Component;
END_VAR
END_METHOD

METHOD DeregisterCyclic : RegistrationResult
VAR_INPUT
	Cyclic : I_Cyclic;
END_VAR
END_METHOD

METHOD DeregisterInitialize : RegistrationResult
VAR_INPUT
	Initializable : I_Initializable;
END_VAR
END_METHOD

METHOD RegisterComponent  : RegistrationResult
VAR_INPUT
	Component : I_Component;
END_VAR
END_METHOD

METHOD RegisterCyclic  : RegistrationResult
VAR_INPUT
	Cyclic : I_Cyclic;
END_VAR
END_METHOD

METHOD RegisterInitialize  : RegistrationResult
VAR_INPUT
	Initializable : I_Initializable;
END_VAR
END_METHOD

END_INTERFACE

// _Internal/Cyclic/Interface/I_Cyclic
INTERFACE I_Cyclic EXTENDS I_Base

METHOD CyclicLogic
VAR_INPUT
END_VAR
END_METHOD

END_INTERFACE

// _Internal/Component/ComponentCollection
FUNCTION_BLOCK ComponentCollection
VAR_GENERIC CONSTANT
	MaxCount : UDINT := 10;
END_VAR IMPLEMENTS I_ComponentCollection
VAR
	Components	   : ARRAY[0..MaxCount] OF I_Component;
	ComponentCount : UDINT;
	NullComponent  : NullComponent('Null Component');
END_VAR

METHOD Accept
VAR_INPUT
	Visitor : I_ComponentVisitor;
END_VAR

VAR
	i : UDINT;
END_VAR
FOR i := 0 TO MaxCount DO
	IF Components[i] = 0 THEN
		EXIT;
	END_IF

	Components[i].Accept(Visitor);
END_FOR
END_METHOD

METHOD AddComponent : RegistrationResult
VAR_INPUT
	Component : I_Component;
END_VAR

VAR
	i : UDINT;
	Registered : BOOL;
END_VAR
IF Component = 0 THEN
	AddComponent := RegistrationResult.NullReference;
	RETURN;
END_IF

IF ComponentCount >= MaxCount THEN
	AddComponent := RegistrationResult.TooManyComponents;
	RETURN;
END_IF

FOR i := 0 TO MaxCount DO
	IF Components[i] = Component THEN
		Registered := TRUE;
	END_IF
END_FOR

IF Registered THEN
	AddComponent := RegistrationResult.AlreadyAdded;
	RETURN;
END_IF

FOR i := 0 TO MaxCount DO
	IF Components[i] = 0 THEN
		Components[i] := Component;
		ComponentCount := ComponentCount + 1;
		EXIT;
	END_IF
END_FOR
END_METHOD

{attribute 'monitoring' := 'call'}
PROPERTY Count : UDINT
GET
Count := TO_UDINT(ComponentCount);
END_GET
END_PROPERTY

METHOD GetAtIndex : I_Component
VAR_INPUT
	Index : UDINT;
END_VAR
IF Index > Count THEN
	GetAtIndex := NullComponent;
	RETURN;
END_IF

IF Index < 0 THEN
	GetAtIndex := NullComponent;
	RETURN;
END_IF

IF Components[Index] <> 0 THEN
	GetAtIndex := Components[Index];
ELSE
	GetAtIndex := NullComponent;
END_IF
END_METHOD

METHOD GetComponentByName : I_Component
VAR_INPUT
	Name : T_MaxString;
END_VAR

VAR
	i : UDINT;
END_VAR
FOR i := 0 TO MaxCount DO
	IF Components[i] = 0 THEN
		EXIT;
	END_IF

	IF Components[i].Name = Name THEN
		GetComponentByName := Components[i];
		EXIT;
	END_IF
END_FOR
END_METHOD

METHOD RemoveComponent : RegistrationResult
VAR_INPUT
	Component : I_Component;
END_VAR

VAR
	i : UDINT;
	PresentInCollection : BOOL;
END_VAR
IF Component = 0 THEN
	RemoveComponent := RegistrationResult.NullReference;
	RETURN;
END_IF

IF ComponentCount = 0 THEN
	RemoveComponent := RegistrationResult.CollectionEmpty;
	RETURN;
END_IF

FOR i := 0 TO MaxCount DO
	IF Components[i] = Component THEN
		PresentInCollection := TRUE;
	END_IF
END_FOR

IF NOT PresentInCollection THEN
	RemoveComponent := RegistrationResult.NotFoundInCollection;
	RETURN;
END_IF

FOR i := 0 TO MaxCount DO
	IF Components[i] = Component THEN
		ComponentCount := ComponentCount - 1;
		IF i < MaxCount THEN
			MEMMOVE(ADR(Components[i]), ADR(Components[i + 1]), (MaxCount - i) * SIZEOF(Component));
		ELSE
			Components[MaxCount] := 0;
		END_IF
		EXIT;
	END_IF
END_FOR
END_METHOD

END_FUNCTION_BLOCK

// _Internal/Null/NullComponent
FUNCTION_BLOCK NullComponent EXTENDS Component
VAR
END_VAR

END_FUNCTION_BLOCK

// _Internal/Cyclic/CyclicRunner
FUNCTION_BLOCK CyclicRunner
VAR_GENERIC CONSTANT
	MaxCount : UDINT := 10;
END_VAR

VAR
	Callees		: ARRAY[0..MaxCount] OF I_Cyclic;
	CalleeCount : UDINT;
END_VAR

METHOD AddCallee : RegistrationResult
VAR_INPUT
	Callee : I_Cyclic;
END_VAR

VAR
	i : UDINT;
	Registered : BOOL;
END_VAR
IF Callee = 0 THEN
	AddCallee := RegistrationResult.NullReference;
	RETURN;
END_IF

IF CalleeCount >= MaxCount THEN
	AddCallee := RegistrationResult.TooManyComponents;
	RETURN;
END_IF

FOR i := 0 TO MaxCount DO
	IF Callees[i] = Callee THEN
		Registered := TRUE;
	END_IF
END_FOR

IF Registered THEN
	AddCallee := RegistrationResult.AlreadyAdded;
	RETURN;
END_IF

FOR i := 0 TO MaxCount DO
	IF Callees[i] = 0 THEN
		Callees[i] := Callee;
		CalleeCount := CalleeCount + 1;
		EXIT;
	END_IF
END_FOR
END_METHOD

METHOD CallAll
VAR_INST
	Logged : BOOL;
END_VAR

VAR
	i	   : UDINT;
	Callee : I_Cyclic;
END_VAR
FOR i := 0 TO MaxCount DO
	IF Callees[i] = 0 THEN
		RETURN;
	END_IF

	Callees[i].CyclicLogic();
END_FOR

IF NOT Logged THEN
	Logged := TRUE;
	Trace.LogMessage('Cyclic Runner', 'Collection is full. Review library parameters and code to ensure proper setup.');
END_IF
END_METHOD

METHOD RemoveCallee : RegistrationResult
VAR_INPUT
	Callee : I_Cyclic;
END_VAR

VAR
	i : UDINT;
	PresentInCollection : BOOL;
END_VAR
IF Callee = 0 THEN
	RemoveCallee := RegistrationResult.NullReference;
	RETURN;
END_IF

IF CalleeCount = 0 THEN
	RemoveCallee := RegistrationResult.CollectionEmpty;
	RETURN;
END_IF

FOR i := 0 TO MaxCount DO
	IF Callees[i] = Callee THEN
		PresentInCollection := TRUE;
	END_IF
END_FOR

IF NOT PresentInCollection THEN
	RemoveCallee := RegistrationResult.NotFoundInCollection;
	RETURN;
END_IF

FOR i := 0 TO MaxCount DO
	IF Callees[i] = Callee THEN
		CalleeCount := CalleeCount - 1;
		IF i < MaxCount THEN
			MEMMOVE(ADR(Callees[i]), ADR(Callees[i + 1]), (MaxCount - i) * SIZEOF(Callee));
		ELSE
			Callees[MaxCount] := 0;
		END_IF
		EXIT;
	END_IF
END_FOR
END_METHOD

END_FUNCTION_BLOCK

// _Internal/Events/TcEventClassArguments
FUNCTION_BLOCK TcEventClassArguments IMPLEMENTS I_EventArguments
VAR
	pArgumentEvent : POINTER TO FB_TcAlarm;
END_VAR

METHOD AddString : I_EventArguments
VAR_INPUT
	Argument : STRING;
END_VAR
IF pArgumentEvent <> 0 THEN
	pArgumentEvent^.ipArguments.AddString(Argument);
END_IF

AddString := THIS^;
END_METHOD

METHOD Clear : I_EventArguments
IF pArgumentEvent <> 0 THEN
	pArgumentEvent^.ipArguments.Clear();
END_IF

Clear := THIS^;
END_METHOD

PROPERTY Event : POINTER TO FB_TcAlarm
SET
pArgumentEvent := Event;
END_SET
END_PROPERTY

END_FUNCTION_BLOCK

// Events/Interface/I_EventArguments
INTERFACE I_EventArguments EXTENDS I_Base

METHOD AddString : I_EventArguments
VAR_INPUT
	Argument : STRING;
END_VAR
END_METHOD

METHOD Clear : I_EventArguments
VAR_INPUT
END_VAR
END_METHOD

END_INTERFACE

// _Internal/Initialize/Initializer
FUNCTION_BLOCK Initializer
VAR_GENERIC CONSTANT
	MaxCount : UDINT := 10;
END_VAR

VAR
	Initializable : ARRAY[0..MaxCount] OF I_Initializable;
	InitializableCount : UDINT;
	NotInitialized : I_Initializable;
END_VAR

METHOD AddInitialize : RegistrationResult
VAR_INPUT
	Initialize : I_Initializable;
END_VAR

VAR
	i : UDINT;
	Registered : BOOL;
END_VAR
IF Initialize = 0 THEN
	AddInitialize := RegistrationResult.NullReference;
	RETURN;
END_IF

IF InitializableCount >= MaxCount THEN
	AddInitialize := RegistrationResult.TooManyComponents;
	RETURN;
END_IF

FOR i := 0 TO MaxCount DO
	IF Initializable[i] = Initialize THEN
		Registered := TRUE;
	END_IF
END_FOR

IF Registered THEN
	AddInitialize := RegistrationResult.AlreadyAdded;
	RETURN;
END_IF

FOR i := 0 TO MaxCount DO
	IF Initializable[i] = 0 THEN
		Initializable[i] := Initialize;
		InitializableCount := InitializableCount + 1;
		EXIT;
	END_IF
END_FOR
END_METHOD

{attribute 'monitoring' := 'call'}
PROPERTY Initialized : BOOL
GET
VAR
	i		   : UDINT;
END_VAR
Initialized	   := TRUE;
NotInitialized := 0;
FOR i := 0 TO MaxCount DO
	IF Initializable[i] = 0 THEN
		EXIT;
	END_IF

	IF NOT Initializable[i].Initialized THEN
		NotInitialized := Initializable[i];
		Initialized	   := FALSE;
	END_IF
END_FOR
END_GET
END_PROPERTY

METHOD Initializing
VAR_INST
	Logged : BOOL;
END_VAR

VAR
	i		   : UDINT;
	Initialize : I_Initializable;
END_VAR
FOR i := 0 TO MaxCount DO
	IF Initializable[i] = 0 THEN
		RETURN;
	END_IF

	Initializable[i].Initialize();
END_FOR

IF NOT Logged THEN
	Logged := TRUE;
	Trace.LogMessage('Initializer', 'Collection is full. Review library parameters and code to ensure proper setup.');
END_IF
END_METHOD

METHOD RemoveInitialize : RegistrationResult
VAR_INPUT
	Initialize : I_Initializable;
END_VAR

VAR
	i : UDINT;
	PresentInCollection : BOOL;
END_VAR
IF Initialize = 0 THEN
	RemoveInitialize := RegistrationResult.NullReference;
	RETURN;
END_IF

IF InitializableCount = 0 THEN
	RemoveInitialize := RegistrationResult.CollectionEmpty;
	RETURN;
END_IF

FOR i := 0 TO MaxCount DO
	IF Initializable[i] = Initialize THEN
		PresentInCollection := TRUE;
	END_IF
END_FOR

IF NOT PresentInCollection THEN
	RemoveInitialize := RegistrationResult.NotFoundInCollection;
	RETURN;
END_IF

FOR i := 0 TO MaxCount DO
	IF Initializable[i] = Initialize THEN
		InitializableCount := InitializableCount - 1;
		IF i < MaxCount THEN
			MEMMOVE(ADR(Initializable[i]), ADR(Initializable[i + 1]), (MaxCount - i) * SIZEOF(Initialize));
		ELSE
			Initializable[MaxCount] := 0;
		END_IF

		EXIT;
	END_IF
END_FOR
END_METHOD

END_FUNCTION_BLOCK

// _Internal/List/Interface/I_List
INTERFACE I_List EXTENDS I_Collection

METHOD ContainsItem : BOOL
VAR_INPUT
	Item : I_Base;
	;
END_VAR
END_METHOD

METHOD GetAtIndex : I_Base
VAR_INPUT
	Index : UDINT;
END_VAR
END_METHOD

METHOD InsertAtIndex : BOOL
VAR_INPUT
	Item  : I_Base;
	Index : UDINT;
END_VAR
END_METHOD

METHOD RemoveAtIndex
VAR_INPUT
	Index : UDINT;
END_VAR
END_METHOD

END_INTERFACE

// _Internal/List/List
FUNCTION_BLOCK List
VAR_GENERIC CONSTANT
	ListSize : UDINT := 2;
END_VAR
EXTENDS Collection<ListSize> IMPLEMENTS I_List
VAR
	_ListCount : UDINT := 0;
END_VAR

METHOD AddItem
VAR_INPUT
	Item : I_Base;
END_VAR
SUPER^.AddItem(Item);
CountListItems();
END_METHOD

METHOD Clear
SUPER^.Clear();
CountListItems();
END_METHOD

METHOD RemoveItem
VAR_INPUT
	Item : I_Base;
END_VAR

VAR
	pItem		 : POINTER TO I_Base;
	pItemNext	 : POINTER TO I_Base;
	i			 : UDINT;
	removedItems : UDINT;
END_VAR
IF _Count = 0 THEN
	Trace.LogMessage(InstancePath, 'No Items found in this Collection!');
	RETURN;
END_IF

IF Item = 0 THEN
	Trace.LogMessage(InstancePath, 'Item to remove needs to be valid interface!');
	RETURN;
END_IF

FOR i := 0 TO (_Count - 1) DO
	IF _Data[i] = Item THEN
		_Data[i]	 := 0;
		removedItems := removedItems + 1;
	END_IF
END_FOR

IF _Count > 1 THEN
	FOR i := 0 TO (_Count - 2) DO
		IF _Data[i] = 0 AND _Data[i + 1] <> 0 THEN
			_Data[i]	 := _Data[i + 1];
			_Data[i + 1] := 0;
		END_IF
	END_FOR
END_IF

CountListItems();
_Count := _Count - removedItems;
END_METHOD

METHOD PRIVATE CountListItems
VAR
	i	  : UDINT;
	pItem : POINTER TO I_Base;
END_VAR
IF _Count = 0 THEN
	_ListCount := 0;
	RETURN;
END_IF

_ListCount := 0;
FOR i := 0 TO (_Count - 1) DO
	IF _Data[i] <> 0 THEN
		_ListCount := _ListCount + 1;
	END_IF
END_FOR
END_METHOD

METHOD ContainsItem : BOOL
VAR_INPUT
	Item : I_Base;
END_VAR

VAR
	i	  : UDINT;
	pItem : POINTER TO I_Base;
END_VAR
IF Item = 0 THEN
	Trace.LogMessage(InstancePath, 'Item is not a valid interface!');
	RETURN;
END_IF

IF _ListCount = 0 THEN
	RETURN;
END_IF

FOR i := 0 TO (_ListCount - 1) DO
	IF _Data[i] = Item AND _Data[i] <> 0 THEN
		ContainsItem := TRUE;
		RETURN;
	END_IF
END_FOR
END_METHOD

{attribute 'monitoring' := 'call'}
PROPERTY Count : UDINT
GET
Count := _ListCount;
END_GET
END_PROPERTY

METHOD GetAtIndex : I_Base
VAR_INPUT
	Index : UDINT;
END_VAR

VAR
	pItem : POINTER TO I_Base;
END_VAR
IF Count = 0 THEN
	Trace.LogMessage(InstancePath, 'No Items found in this List!');
	RETURN;
END_IF

IF Index > (_Count - 1) THEN
	Trace.LogMessage(InstancePath, 'Index does not exist in List!');
	RETURN;
END_IF

GetAtIndex := _Data[Index];
END_METHOD

METHOD InsertAtIndex : BOOL
VAR_INPUT
	Item  : I_Base;
	Index : UDINT;
END_VAR

VAR
	pItem	  : POINTER TO I_Base;
	pItemNext : POINTER TO I_Base;
	i		  : UDINT;
END_VAR
IF Index > _Count THEN
	InsertAtIndex := FALSE;
	RETURN;
END_IF

_Count := (_Count + 1);
FOR i := _Count TO Index + 1 BY -1 DO
	_Data[i] := _Data[i - 1];
END_FOR

_Data[Index] := Item;
CountListItems();
END_METHOD

METHOD RemoveAtIndex
VAR_INPUT
	Index : UDINT;
END_VAR

VAR
	pItem : POINTER TO I_Base;
END_VAR
IF Count = 0 THEN
	Trace.LogMessage(InstancePath, 'No Items found in this List!');
	RETURN;
END_IF

IF Index > (_Count - 1) THEN
	Trace.LogMessage(InstancePath, 'Index does not exist in List!');
	RETURN;
END_IF

MEMMOVE(ADR(_Data[Index]), ADR(_Data[Index + 1]), (_Count - Index - 1) * SIZEOF(PVOID));
_Count := _Count - 1;

//pItem  := Collection.pBuffer + (Index * SIZEOF(PVOID));
CountListItems();
END_METHOD

END_FUNCTION_BLOCK

// _Internal/Module/Interface/I_ContainModules
INTERFACE I_ContainModules EXTENDS I_Base

METHOD DeregisterCyclic : RegistrationResult
VAR_INPUT
	Cyclic : I_Cyclic;
END_VAR
END_METHOD

METHOD DeregisterInitialize : RegistrationResult
VAR_INPUT
	Initializable : I_Initializable;
END_VAR
END_METHOD

METHOD DeregisterModule : RegistrationResult
VAR_INPUT
	Module : I_Module;
END_VAR
END_METHOD

PROPERTY Modules : I_ModuleCollection
GET
END_GET
END_PROPERTY

METHOD RegisterCyclic  : RegistrationResult
VAR_INPUT
	Cyclic : I_Cyclic;
END_VAR
END_METHOD

METHOD RegisterInitialize  : RegistrationResult
VAR_INPUT
	Initializable : I_Initializable;
END_VAR
END_METHOD

METHOD RegisterModule  : RegistrationResult
VAR_INPUT
	Module : I_Module;
END_VAR
END_METHOD

END_INTERFACE

// Module/Module
FUNCTION_BLOCK ABSTRACT Module IMPLEMENTS I_Module, I_Cyclic, I_Initializable
VAR
	_Name				: T_MaxString;
	ModuleInitialized	: BOOL;
	CyclicRunner		: CyclicRunner<ApplicationBaseParameter.MaxCountInCollections>;
	ComponentCollection : ComponentCollection<ApplicationBaseParameter.MaxCountInCollections>;
	ModuleCollection	: ModuleCollection<ApplicationBaseParameter.MaxCountInCollections>;
	Initializer			: Initializer<ApplicationBaseParameter.MaxCountInCollections>;
END_VAR

//FB_Init is always available implicitly and it is used primarily for initialization.

//The return value is not evaluated. For a specific influence, you can also declare the

//methods explicitly and provide additional code there with the standard initialization

//code. You can evaluate the return value.
METHOD FB_Init : BOOL
VAR_INPUT
	bInitRetains : BOOL; // TRUE: the retain variables are initialized (reset warm / reset cold)
	bInCopyCode	 : BOOL; // TRUE: the instance will be copied to the copy code afterward (online change)   
	Name		 : T_MaxString;
END_VAR
_Name := Name;
END_METHOD

METHOD CyclicLogic
OnCyclicCall();
CyclicRunner.CallAll();
END_METHOD

METHOD ABSTRACT OnCyclicCall
VAR_INPUT
END_VAR
END_METHOD

METHOD DeregisterComponent : RegistrationResult
VAR_INPUT
	Component : I_Component;
END_VAR
DeregisterComponent := ComponentCollection.RemoveComponent(Component);
END_METHOD

METHOD DeregisterCyclic : RegistrationResult
VAR_INPUT
	Cyclic : I_Cyclic;
END_VAR
DeregisterCyclic := CyclicRunner.RemoveCallee(Cyclic);
END_METHOD

METHOD DeregisterInitialize : RegistrationResult
VAR_INPUT
	Initializable : I_Initializable;
END_VAR
DeregisterInitialize := Initializer.RemoveInitialize(Initializable);
END_METHOD

METHOD DeregisterModule : RegistrationResult
VAR_INPUT
	Module : I_Module;
END_VAR
DeregisterModule := ModuleCollection.RemoveModule(Module);
END_METHOD

METHOD DeregisterWithParent
VAR_INPUT
	Parent : I_ContainModules;
END_VAR
Parent.DeregisterModule(THIS^);
Parent.DeregisterCyclic(THIS^);
Parent.DeregisterInitialize(THIS^);
END_METHOD

METHOD Initialize
IF NOT ModuleInitialized THEN
	Initializing();
	RETURN;
END_IF

Initializer.Initializing();
END_METHOD

{attribute 'monitoring' := 'call'}
PROPERTY Initialized : BOOL
GET
Initialized := ModuleInitialized AND Initializer.Initialized;
END_GET
SET
ModuleInitialized := Initialized;
END_SET
END_PROPERTY

(* This Module will be done initialize when ModuleInitialized := TRUE;, subequently all subitems will be called to be initialized *)
METHOD ABSTRACT Initializing
// ModuleInitialized := TRUE;
END_METHOD

METHOD RegisterComponent : RegistrationResult
VAR_INPUT
	Component : I_Component;
END_VAR
RegisterComponent := ComponentCollection.AddComponent(Component);
END_METHOD

METHOD RegisterCyclic : RegistrationResult
VAR_INPUT
	Cyclic : I_Cyclic;
END_VAR
RegisterCyclic := CyclicRunner.AddCallee(Cyclic);
END_METHOD

METHOD RegisterInitialize : RegistrationResult
VAR_INPUT
	Initializable : I_Initializable;
END_VAR
RegisterInitialize := Initializer.AddInitialize(Initializable);
END_METHOD

METHOD RegisterModule : RegistrationResult
VAR_INPUT
	Module : I_Module;
END_VAR
RegisterModule := ModuleCollection.AddModule(Module);
END_METHOD

METHOD RegisterWithParent
VAR_INPUT
	Parent : I_ContainModules;
END_VAR
Parent.RegisterModule(THIS^);
Parent.RegisterCyclic(THIS^);
Parent.RegisterInitialize(THIS^);
END_METHOD

METHOD ResetComponents : BOOL
VAR_INST
	ResetComponentsVisitor : ResetComponentsVisitor;
END_VAR
ResetComponentsVisitor.Reset(THIS^);
ResetComponents := NOT ResetComponentsVisitor.Error AND NOT ResetComponentsVisitor.Busy;
END_METHOD

METHOD ResetModules : BOOL
VAR_INST
	ResetModulesVisitor : ResetModulesVisitor;
END_VAR
ResetModulesVisitor.Reset(THIS^);
ResetModules := NOT ResetModulesVisitor.Error AND NOT ResetModulesVisitor.Busy;
END_METHOD

METHOD Accept
VAR_INPUT
	Visitor : I_ModuleVisitor;
END_VAR
Visitor.VisitModule(THIS^);
END_METHOD

PROPERTY Components : I_ComponentCollection
GET
Components := ComponentCollection;
END_GET
END_PROPERTY

PROPERTY Modules : I_ModuleCollection
GET
Modules := ModuleCollection;
END_GET
END_PROPERTY

{attribute 'monitoring' := 'call'}
PROPERTY Name : T_MaxString
GET
Name := _Name;
END_GET
SET
_Name := Name;
END_SET
END_PROPERTY

END_FUNCTION_BLOCK

// Module/Interface/I_Module
INTERFACE I_Module EXTENDS I_ContainComponents, I_ContainModules, I_Base

METHOD Accept
VAR_INPUT
	Visitor : I_ModuleVisitor;
END_VAR
END_METHOD

METHOD DeregisterWithParent
VAR_INPUT
	Parent : I_ContainModules;
END_VAR
END_METHOD

{attribute 'monitoring' := 'call'}
PROPERTY Name : T_MaxString
GET
END_GET
END_PROPERTY

METHOD RegisterWithParent
VAR_INPUT
	Parent : I_ContainModules;
END_VAR
END_METHOD

METHOD ResetComponents : BOOL
END_METHOD

METHOD ResetModules : BOOL
END_METHOD

END_INTERFACE

// Module/Interface/I_ModuleVisitor
INTERFACE I_ModuleVisitor

METHOD VisitModule
VAR_INPUT
	Module : I_Module;
END_VAR
END_METHOD

END_INTERFACE

// _Internal/Module/ModuleCollection
FUNCTION_BLOCK ModuleCollection
VAR_GENERIC CONSTANT
	MaxCount : UDINT := 10;
END_VAR IMPLEMENTS I_ModuleCollection
VAR
	Modules		: ARRAY[0..MaxCount] OF I_Module;
	ModuleCount : UDINT;
	NullModule	: NullModule('Null Module');
END_VAR

METHOD Accept
VAR_INPUT
	Visitor : I_ModuleVisitor;
END_VAR

VAR
	i : UDINT;
END_VAR
FOR i := 0 TO MaxCount DO
	IF Modules[i] = 0 THEN
		EXIT;
	END_IF

	Modules[i].Accept(Visitor);
END_FOR
END_METHOD

METHOD AddModule : RegistrationResult
VAR_INPUT
	Module : I_Module;
END_VAR

VAR
	i : UDINT;
	Registered : BOOL;
END_VAR
IF Module = 0 THEN
	AddModule := RegistrationResult.NullReference;
	RETURN;
END_IF

IF ModuleCount >= MaxCount THEN
	AddModule := RegistrationResult.TooManyComponents;
	RETURN;
END_IF

FOR i := 0 TO MaxCount DO
	IF Modules[i] = Module THEN
		Registered := TRUE;
	END_IF
END_FOR

IF Registered THEN
	AddModule := RegistrationResult.AlreadyAdded;
	RETURN;
END_IF

FOR i := 0 TO MaxCount DO
	IF Modules[i] = 0 THEN
		Modules[i] := Module;
		ModuleCount := ModuleCount + 1;
		EXIT;
	END_IF
END_FOR
END_METHOD

{attribute 'monitoring' := 'call'}
PROPERTY Count : UDINT
GET
Count := TO_UDINT(ModuleCount);
END_GET
END_PROPERTY

METHOD GetAtIndex : I_Module
VAR_INPUT
	Index : UDINT;
END_VAR
IF Index > Count THEN
	GetAtIndex := NullModule;
	RETURN;
END_IF

IF Index < 0 THEN
	GetAtIndex := NullModule;
	RETURN;
END_IF

IF Modules[Index] <> 0 THEN
	GetAtIndex := Modules[Index];
ELSE
	GetAtIndex := NullModule;
END_IF
END_METHOD

METHOD GetModuleByName : I_Module
VAR_INPUT
	Name : T_MaxString;
END_VAR

VAR
	i : UDINT;
END_VAR
FOR i := 0 TO MaxCount DO
	IF Modules[i] = 0 THEN
		EXIT;
	END_IF

	IF Modules[i].Name = Name THEN
		GetModuleByName := Modules[i];
		EXIT;
	END_IF
END_FOR
END_METHOD

METHOD RemoveModule : RegistrationResult
VAR_INPUT
	Module : I_Module;
END_VAR

VAR
	i : UDINT;
	PresentInCollection : BOOL;
END_VAR
IF Module = 0 THEN
	RemoveModule := RegistrationResult.NullReference;
	RETURN;
END_IF

IF ModuleCount = 0 THEN
	RemoveModule := RegistrationResult.CollectionEmpty;
	RETURN;
END_IF

FOR i := 0 TO MaxCount DO
	IF Modules[i] = Module THEN
		PresentInCollection := TRUE;
	END_IF
END_FOR

IF NOT PresentInCollection THEN
	RemoveModule := RegistrationResult.NotFoundInCollection;
	RETURN;
END_IF

FOR i := 0 TO MaxCount DO
	IF Modules[i] = Module THEN
		IF i < MaxCount THEN
			MEMMOVE(ADR(Modules[i]), ADR(Modules[i + 1]), (MaxCount - i) * SIZEOF(Module));
		ELSE
			Modules[MaxCount] := 0;
		END_IF

		EXIT;
	END_IF
END_FOR
END_METHOD

END_FUNCTION_BLOCK

// _Internal/Module/Interface/I_ModuleCollection
INTERFACE I_ModuleCollection EXTENDS I_Base

METHOD Accept
VAR_INPUT
	Visitor : I_ModuleVisitor;
END_VAR
END_METHOD

{attribute 'monitoring' := 'call'}
PROPERTY Count : UDINT
GET
END_GET
END_PROPERTY

METHOD GetAtIndex : I_Module
VAR_INPUT
	Index : UDINT;
END_VAR
END_METHOD

METHOD GetModuleByName : I_Module
VAR_INPUT
	Name : T_MaxString;
END_VAR
END_METHOD

END_INTERFACE

// _Internal/Null/NullModule
FUNCTION_BLOCK NullModule IMPLEMENTS I_Module
VAR
    _Name : T_MaxString;
END_VAR

METHOD Accept
VAR_INPUT
	Visitor	: I_ModuleVisitor;
END_VAR
END_METHOD

PROPERTY Components : I_ComponentCollection
GET
END_GET
END_PROPERTY

METHOD DeregisterComponent : RegistrationResult
VAR_INPUT
	Component	: I_Component;
END_VAR
END_METHOD

METHOD DeregisterCyclic : RegistrationResult
VAR_INPUT
	Cyclic	: I_Cyclic;
END_VAR
END_METHOD

METHOD DeregisterInitialize : RegistrationResult
VAR_INPUT
	Initializable	: I_Initializable;
END_VAR
END_METHOD

METHOD DeregisterModule : RegistrationResult
VAR_INPUT
	Module	: I_Module;
END_VAR
END_METHOD

METHOD DeregisterWithParent
VAR_INPUT
	Parent	: I_ContainModules;
END_VAR
END_METHOD

//FB_Init is always available implicitly and it is used primarily for initialization.

//The return value is not evaluated. For a specific influence, you can also declare the

//methods explicitly and provide additional code there with the standard initialization

//code. You can evaluate the return value.
METHOD FB_Init : BOOL
VAR_INPUT
	bInitRetains : BOOL; // TRUE: the retain variables are initialized (reset warm / reset cold)
	bInCopyCode	 : BOOL; // TRUE: the instance will be copied to the copy code afterward (online change)   
	Name		 : T_MaxString;
END_VAR
_Name := Name;
END_METHOD

PROPERTY Modules : I_ModuleCollection
GET
END_GET
END_PROPERTY

{attribute 'monitoring' := 'call'}
PROPERTY Name : T_MaxString
GET
Name := _Name;
END_GET
SET
_Name := Name;
END_SET
END_PROPERTY

METHOD RegisterComponent : RegistrationResult
VAR_INPUT
	Component	: I_Component;
END_VAR
END_METHOD

METHOD RegisterCyclic : RegistrationResult
VAR_INPUT
	Cyclic	: I_Cyclic;
END_VAR
END_METHOD

METHOD RegisterInitialize : RegistrationResult
VAR_INPUT
	Initializable	: I_Initializable;
END_VAR
END_METHOD

METHOD RegisterModule : RegistrationResult
VAR_INPUT
	Module	: I_Module;
END_VAR
END_METHOD

METHOD RegisterWithParent
VAR_INPUT
	Parent	: I_ContainModules;
END_VAR
END_METHOD

METHOD ResetComponents : BOOL
END_METHOD

METHOD ResetModules : BOOL
END_METHOD

END_FUNCTION_BLOCK

// Visitors/Reset/ResetComponentsVisitor
FUNCTION_BLOCK ResetComponentsVisitor IMPLEMENTS I_ComponentVisitor, I_TaskResult
VAR
	{attribute 'hide'}
	Resettable : I_Resettable;
	{attribute 'hide'}
	Result : I_TaskResult;
	{attribute 'hide'}
	_Busy : BOOL;
	{attribute 'hide'}
	_Error : BOOL;
	{attribute 'hide'}
	_ErrorId	   : UDINT;
	ErrorComponent : I_Component;
END_VAR

{attribute 'monitoring' := 'call'}
PROPERTY Busy : BOOL
GET
Busy := _Busy;
END_GET
END_PROPERTY

{attribute 'monitoring' := 'call'}
PROPERTY Error : BOOL
GET
Error := _Error;
END_GET
END_PROPERTY

{attribute 'monitoring' := 'call'}
PROPERTY ErrorId : UDINT
GET
ErrorID := _ErrorID;
END_GET
END_PROPERTY

METHOD Reset
VAR_INPUT
	Module : I_Module;
END_VAR
_Error	 := FALSE;
_ErrorId := 0;
_Busy	 := FALSE;
Module.Components.Accept(THIS^);
END_METHOD

METHOD VisitComponent
VAR_INPUT
	Component : I_Component;
END_VAR
IF __QUERYINTERFACE(Component, Resettable) THEN
	Resettable.Reset();
END_IF

IF __QUERYINTERFACE(Component, Result) THEN
	IF Result.Error THEN
		ErrorComponent := Component;
		_Error		   := TRUE;
		_ErrorId	   := Result.ErrorId;
	END_IF

	IF Result.Busy THEN
		_Busy := TRUE;
	END_IF
END_IF
END_METHOD

END_FUNCTION_BLOCK

// Visitors/Reset/ResetModulesVisitor
FUNCTION_BLOCK ResetModulesVisitor IMPLEMENTS I_ModuleVisitor, I_TaskResult
VAR
	{attribute 'hide'}
	Resettable : I_Resettable;
	{attribute 'hide'}
	Result : I_TaskResult;
	{attribute 'hide'}
	_Busy : BOOL;
	{attribute 'hide'}
	_Error : BOOL;
	{attribute 'hide'}
	_ErrorId	: UDINT;
	ErrorModule : I_Module;
END_VAR

{attribute 'monitoring' := 'call'}
PROPERTY Busy : BOOL
GET
Busy := _Busy;
END_GET
END_PROPERTY

{attribute 'monitoring' := 'call'}
PROPERTY Error : BOOL
GET
Error := _Error;
END_GET
END_PROPERTY

{attribute 'monitoring' := 'call'}
PROPERTY ErrorId : UDINT
GET
ErrorID := _ErrorID;
END_GET
END_PROPERTY

METHOD Reset
VAR_INPUT
	Module : I_Module;
END_VAR
_Error	 := FALSE;
_ErrorId := 0;
_Busy	 := FALSE;
Module.Modules.Accept(THIS^);
END_METHOD

METHOD VisitModule
VAR_INPUT
	Module : I_Module;
END_VAR
IF __QUERYINTERFACE(Module, Resettable) THEN
	Resettable.Reset();
END_IF

IF __QUERYINTERFACE(Module, Result) THEN
	IF Result.Error THEN
		ErrorModule := Module;
		_Error		:= TRUE;
		_ErrorId	:= Result.ErrorId;
	END_IF

	IF Result.Busy THEN
		_Busy := TRUE;
	END_IF
END_IF
END_METHOD

END_FUNCTION_BLOCK

// _Internal/MotionTasks/AX5000/MotionTask_AX5000AmpToNm
FUNCTION_BLOCK MotionTask_AX5000AmpToNm EXTENDS MotionTask
VAR
	i					   : INT;
	SequenceState		   : DINT := -10;
	RawConfigChPeakCurrent : UDINT;					// Configured Channel Peak Current  ( raw )
	ConfigChPeakCurrent	   : LREAL;					// Configured Channel Peak Current  ( units := A )
	MotorConsType		   : WORD;					// Motor construction type          ( raw )
	MotorType			   : BOOL;					// Motor construction type          ( units := 0 = Rotary, 1 = Linear ) 
	RawContStallTorque	   : UDINT;					// Motor continuous stall torque    ( raw )
	ContStallTorque		   : LREAL;					// Motor continuous stall torque    ( units := Nm )
	ContStallTorqueEx	   : LREAL;					// Motor continuous stall torque    ( units := Nm ) - extended slope   
	RawPeakTorque		   : UDINT;					// Motor peak torque                ( raw )
	PeakTorque			   : LREAL;					// Motor peak torque                ( units := Nm )
	RawContStallForce	   : UDINT;					// Motor continuous stall force     ( raw )
	ContStallForce		   : LREAL;					// Motor continuous stall force     ( units := N )
	ContStallForceEx	   : LREAL;					// Motor continuous stall force     ( units := N ) - extended slope
	RawPeakForce		   : UDINT;					// Motor peak force                 ( raw )
	PeakForce			   : LREAL;					// Motor peak force                 ( units := N )
	RawContStallCurrent	   : UDINT;					// Motor continuous stall current   ( raw )
	ContStallCurrent	   : LREAL;					// Motor continuous stall current   ( units := A )
	ContStallCurrentEx	   : LREAL;					// Motor continuous stall current   ( units := A ) - extended slope
	RawPeakCurrent		   : UDINT;					// Motor peak current               ( raw )
	PeakCurrent			   : LREAL;					// Motor peak current               ( units := A )
	Scale				   : LREAL;					// Position between array indexes   ( units := % )
	SoERead				   : FB_SoERead;			// Read SoE params from drive
	RawMotorTorqueCurve	   : ST_IDN_P_0_0074_UDINT; // Contents read in from P-0-0074   ( raw )
END_VAR

VAR
	_ErrorId		 : UDINT;			 // 1 = Axis Not Linked, 2 = Failed To Read P-0-0074, 3 = Failed To Read P-0-0092, 4 = Failed To Read P-0-0050, 5 = Failed To Read P-0-0070, 6 = Failed To Read P-0-0126, 7 = Failed To Read S-0-0111
	CalculatedValues : ST_AX5000AmpToNm; // Data read in and calculated from the drive
END_VAR

(*  
Error Ids:
  1 = Axis Not Linked, 
  2 = Failed To Read P-0-0074,
  3 = Failed To Read P-0-0092, 
  4 = Failed To Read P-0-0050, 
  5 = Failed To Read P-0-0070, 
  6 = Failed To Read P-0-0126, 
  7 = Failed To Read S-0-0111 
*)

{attribute 'monitoring' := 'call'}
PROPERTY ActCurrent : LREAL
GET
ActCurrent := CalculatedValues.ActCurrent;
END_GET
END_PROPERTY

{attribute 'monitoring' := 'call'}
PROPERTY ActTorque : LREAL
GET
ActTorque := CalculatedValues.ActTorque;
END_GET
END_PROPERTY

{attribute 'monitoring' := 'call'}
PROPERTY Busy : BOOL
GET
Busy := SequenceState > 0 AND SequenceState <= 100;
END_GET
END_PROPERTY

METHOD CyclicLogic
IF _Axis = 0 THEN
	RETURN;
END_IF

CASE SequenceState OF
	-10: // Initialize
		RawConfigChPeakCurrent := 0;
		ConfigChPeakCurrent	   := 0.0;
		MotorConsType		   := 0;
		MotorType			   := FALSE;
		RawContStallTorque	   := 0;
		ContStallTorque		   := 0.0;
		ContStallTorqueEx	   := 0.0;
		RawPeakTorque		   := 0;
		PeakTorque			   := 0.0;
		RawContStallForce	   := 0;
		ContStallForce		   := 0.0;
		ContStallForceEx	   := 0.0;
		RawPeakForce		   := 0;
		PeakForce			   := 0.0;
		RawContStallCurrent	   := 0;
		ContStallCurrent	   := 0.0;
		ContStallCurrentEx	   := 0.0;
		RawPeakCurrent		   := 0;
		PeakCurrent			   := 0.0;
		Scale				   := 0.0;
		SoERead(Execute := FALSE, Axis := _Axis.Axis);
		MEMSET(ADR(RawMotorTorqueCurve), 16#0, SIZEOF(RawMotorTorqueCurve));
		MEMSET(ADR(CalculatedValues), 16#0, SIZEOF(CalculatedValues));
		IF _Axis.Axis.NcToPlc.AxisId = 0 THEN
			_ErrorId	  := 1;
			SequenceState := 5000;
		ELSE
			SequenceState := SequenceState + 10;
		END_IF

	0:	// Wait for Execute()  
	10: // Read in the value of P-0-0074 ( Motor torque characteristic )
		SoERead(NetId	:= '',
				Idn		:= P_0_IDNs + 74,
				Element := 16#40,
				pDstBuf := ADR(RawMotorTorqueCurve),
				BufLen	:= SIZEOF(RawMotorTorqueCurve),
				Execute := TRUE,
				Axis	:= _Axis.Axis);

		IF NOT SoERead.Busy AND NOT SoERead.Error THEN
			SoERead(Execute := FALSE, Axis := _Axis.Axis);
			FOR i := 0 TO 9 DO // Convert raw values into actual units
				CalculatedValues.Curve.Iq[i] := UDINT_TO_LREAL(RawMotorTorqueCurve.Elements.Iq[i]) / 1000.0;
				CalculatedValues.Curve.M[i]	 := UDINT_TO_LREAL(RawMotorTorqueCurve.Elements.M[i]) / 100.0;
			END_FOR

			SequenceState := SequenceState + 10;
		ELSIF SoERead.Error THEN
			SoERead(Execute := FALSE, Axis := _Axis.Axis);
			_ErrorId	  := 2;
			SequenceState := 5000;
		END_IF

	20: // Read in the value of P-0-0092 ( Configured channel peak current )       
		SoERead(NetId	:= '',
				Idn		:= P_0_IDNs + 92,
				Element := 16#40,
				pDstBuf := ADR(RawConfigChPeakCurrent),
				BufLen	:= SIZEOF(RawConfigChPeakCurrent),
				Execute := TRUE,
				Axis	:= _Axis.Axis);

		IF NOT SoERead.Busy AND NOT SoERead.Error THEN // Convert raw values into actual units
			SoERead(Execute := FALSE, Axis := _Axis.Axis);
			ConfigChPeakCurrent := UDINT_TO_LREAL(RawConfigChPeakCurrent) / 1000.0;
			SequenceState		:= SequenceState + 10;
		ELSIF SoERead.Error THEN
			SoERead(Execute := FALSE, Axis := _Axis.Axis);
			_ErrorId	  := 3;
			SequenceState := 5000;
		END_IF

	30: // Check for valid characteristic curve
		IF RawMotorTorqueCurve.Elements.Iq[9] = 0 THEN
			SequenceState := SequenceState + 10; // Curve is not available
		ELSE
			SequenceState := 1000; // Curve is available
		END_IF

	40: // Read in the value of P-0-0050 ( Motor construction type )       
		SoERead(NetId	:= '',
				Idn		:= P_0_IDNs + 50,
				Element := 16#40,
				pDstBuf := ADR(MotorConsType),
				BufLen	:= SIZEOF(MotorConsType),
				Execute := TRUE,
				Axis	:= _Axis.Axis);

		IF NOT SoERead.Busy AND NOT SoERead.Error THEN
			SoERead(Execute := FALSE, Axis := _Axis.Axis);
			MotorType := MotorConsType.1;
			IF NOT MotorType THEN
				SequenceState := 50; // Rotary
			ELSE
				SequenceState := 70; // Linear
			END_IF
		ELSIF SoERead.Error THEN
			SoERead(Execute := FALSE, Axis := _Axis.Axis);
			_ErrorId	  := 4;
			SequenceState := 5000;
		END_IF

	50: // Read in the value of P-0-0070 ( Motor continuous stall torque )       
		SoERead(NetId	:= '',
				Idn		:= P_0_IDNs + 70,
				Element := 16#40,
				pDstBuf := ADR(RawContStallTorque),
				BufLen	:= SIZEOF(RawContStallTorque),
				Execute := TRUE,
				Axis	:= _Axis.Axis);

		IF NOT SoERead.Busy AND NOT SoERead.Error THEN
			SoERead(Execute := FALSE, Axis := _Axis.Axis);
			ContStallTorque := UDINT_TO_LREAL(RawContStallTorque) / 100.0;
			SequenceState	:= SequenceState + 10;
		ELSIF SoERead.Error THEN
			SoERead(Execute := FALSE, Axis := _Axis.Axis);
			_ErrorId	  := 5;
			SequenceState := 5000;
		END_IF

	60: // Read in the value of P-0-0073 ( Motor peak torque )       
		SoERead(NetId	:= '',
				Idn		:= P_0_IDNs + 73,
				Element := 16#40,
				pDstBuf := ADR(RawPeakTorque),
				BufLen	:= SIZEOF(RawPeakTorque),
				Execute := TRUE,
				Axis	:= _Axis.Axis);

		IF NOT SoERead.Busy AND NOT SoERead.Error THEN
			SoERead(Execute := FALSE, Axis := _Axis.Axis);
			PeakTorque	  := UDINT_TO_LREAL(RawPeakTorque) / 100.0;
			SequenceState := 90;
		ELSIF SoERead.Error THEN
			SoERead(Execute := FALSE, Axis := _Axis.Axis);
			SequenceState := 90;
		END_IF

	70: // Read in the value of P-0-0126 ( Motor continuous stall force )       
		SoERead(NetId	:= '',
				Idn		:= P_0_IDNs + 126,
				Element := 16#40,
				pDstBuf := ADR(RawContStallForce),
				BufLen	:= SIZEOF(RawContStallForce),
				Execute := TRUE,
				Axis	:= _Axis.Axis);

		IF NOT SoERead.Busy AND NOT SoERead.Error THEN
			SoERead(Execute := FALSE, Axis := _Axis.Axis);
			ContStallForce := UDINT_TO_LREAL(RawContStallForce) / 100.0;
			SequenceState  := SequenceState + 10;
		ELSIF SoERead.Error THEN
			SoERead(Execute := FALSE, Axis := _Axis.Axis);
			_ErrorId	  := 6;
			SequenceState := 5000;
		END_IF

	80: // Read in the value of P-0-0128 ( Motor peak force )       
		SoERead(NetId	:= '',
				Idn		:= P_0_IDNs + 128,
				Element := 16#40,
				pDstBuf := ADR(RawPeakForce),
				BufLen	:= SIZEOF(RawPeakForce),
				Execute := TRUE,
				Axis	:= _Axis.Axis);

		IF NOT SoERead.Busy AND NOT SoERead.Error THEN
			SoERead(Execute := FALSE, Axis := _Axis.Axis);
			PeakForce	  := UDINT_TO_LREAL(RawPeakForce) / 100.0;
			SequenceState := SequenceState + 10;
		ELSIF SoERead.Error THEN
			SoERead(Execute := FALSE, Axis := _Axis.Axis);
			SequenceState := SequenceState + 10;
		END_IF

	90: // Read in the value of S-0-0111 ( Motor continuous stall current )       
		SoERead(NetId	:= '',
				Idn		:= S_0_IDNs + 111,
				Element := 16#40,
				pDstBuf := ADR(RawContStallCurrent),
				BufLen	:= SIZEOF(RawContStallCurrent),
				Execute := TRUE,
				Axis	:= _Axis.Axis);

		IF NOT SoERead.Busy AND NOT SoERead.Error THEN
			SoERead(Execute := FALSE, Axis := _Axis.Axis);
			ContStallCurrent := UDINT_TO_LREAL(RawContStallCurrent) / 1000.0;
			SequenceState	 := SequenceState + 10;
		ELSIF SoERead.Error THEN
			SoERead(Execute := FALSE, Axis := _Axis.Axis);
			_ErrorId	  := 7;
			SequenceState := 5000;
		END_IF

	100: // Read in the value of S-0-0109 ( Motor peak current )       
		SoERead(NetId	:= '',
				Idn		:= S_0_IDNs + 109,
				Element := 16#40,
				pDstBuf := ADR(RawPeakCurrent),
				BufLen	:= SIZEOF(RawPeakCurrent),
				Execute := TRUE,
				Axis	:= _Axis.Axis);

		IF NOT SoERead.Busy THEN
			SoERead(Execute := FALSE, Axis := _Axis.Axis);
			PeakCurrent := UDINT_TO_LREAL(RawPeakCurrent) / 1000.0;
			IF NOT MotorType THEN
				IF PeakCurrent = 0 OR PeakTorque = 0 THEN
					SequenceState := 300; // Rotary Motor: Curve not available... peak torque and current missing - Using slope of points 0,0 to P-0-0070 and S-0-0111
				ELSE
					SequenceState := 200; // Rotary Motor: Curve not available - Using linear interpolation of points P-0-0070, P-0-0073, S-0-0111 and S-0-0109
				END_IF
			ELSE
				IF PeakCurrent = 0 OR PeakForce = 0 THEN
					SequenceState := 500; // Linear Motor: Curve not available... peak torque and current missing - Using slope of points 0,0 to P-0-0126 and S-0-0111
				ELSE
					SequenceState := 400; // Linear Motor: Curve not available - Using linear interpolation of points P-0-0126, P-0-0128, S-0-0111 and S-0-0109
				END_IF
			END_IF
		END_IF

	200: // Rotary Motor: Curve not available - Using linear interpolation of points P-0-0070, P-0-0073, S-0-0111 and S-0-0109
		CalculatedValues.ActCurrent := ABS((_Axis.Axis.NcToPlc.ActTorque / 100) * ConfigChPeakCurrent);
		// Convert the actual current in amps to Nm
		IF CalculatedValues.ActCurrent = 0 THEN
			CalculatedValues.ActTorque := 0;
		ELSIF CalculatedValues.ActCurrent > 0 AND CalculatedValues.ActCurrent < ContStallCurrent THEN
			IF ContStallCurrent > 0 THEN
				Scale					   := CalculatedValues.ActCurrent / ContStallCurrent;
				CalculatedValues.ActTorque := Scale * ContStallTorque;
			END_IF
		ELSIF CalculatedValues.ActCurrent >= ContStallCurrent AND CalculatedValues.ActCurrent <= PeakCurrent THEN
			IF (CalculatedValues.ActCurrent - ContStallCurrent) > 0 AND (PeakCurrent - ContStallCurrent) > 0 THEN
				Scale					   := (CalculatedValues.ActCurrent - ContStallCurrent) / (PeakCurrent - ContStallCurrent);
				CalculatedValues.ActTorque := (Scale * (PeakTorque - ContStallTorque) + ContStallTorque);
			END_IF
		END_IF

	300: // Rotary Motor: Curve not available... peak torque and current missing - Using slope of points 0,0 to P-0-0070 and S-0-0111
		CalculatedValues.ActCurrent := ABS((_Axis.Axis.NcToPlc.ActTorque / 100) * ConfigChPeakCurrent);

		// Project slope from continuous stall torque/current
		ContStallCurrentEx := ContStallCurrent * 10.0;
		ContStallTorqueEx  := ContStallTorque * 10.0;
		// Convert the actual current in amps to Nm
		IF CalculatedValues.ActCurrent = 0 THEN
			CalculatedValues.ActTorque := 0;
		ELSIF CalculatedValues.ActCurrent > 0 AND CalculatedValues.ActCurrent <= ContStallCurrentEx THEN
			IF ContStallCurrentEx > 0 THEN
				Scale					   := CalculatedValues.ActCurrent / ContStallCurrentEx;
				CalculatedValues.ActTorque := Scale * ContStallTorqueEx;
			END_IF
		END_IF

	400: // Linear Motor: Curve not available - Using linear interpolation of points P-0-0126, P-0-0128, S-0-0111 and S-0-0109
		CalculatedValues.ActCurrent := ABS((_Axis.Axis.NcToPlc.ActTorque / 100) * ConfigChPeakCurrent);
		// Convert the actual current in amps to Nm
		IF CalculatedValues.ActCurrent = 0 THEN
			CalculatedValues.ActTorque := 0;
		ELSIF CalculatedValues.ActCurrent > 0 AND CalculatedValues.ActCurrent < ContStallCurrent THEN
			IF ContStallCurrent > 0 THEN
				Scale					   := CalculatedValues.ActCurrent / ContStallCurrent;
				CalculatedValues.ActTorque := Scale * ContStallForce;
			END_IF
		ELSIF CalculatedValues.ActCurrent >= ContStallCurrent AND CalculatedValues.ActCurrent <= PeakCurrent THEN
			IF (CalculatedValues.ActCurrent - ContStallCurrent) > 0 AND (PeakCurrent - ContStallCurrent) > 0 THEN
				Scale					   := (CalculatedValues.ActCurrent - ContStallCurrent) / (PeakCurrent - ContStallCurrent);
				CalculatedValues.ActTorque := (Scale * (PeakForce - ContStallForce) + ContStallForce);
			END_IF
		END_IF

	500: // Linear Motor: Curve not available... peak torque and current missing - Using slope of points 0,0 to P-0-0126 and S-0-0111
		CalculatedValues.ActCurrent := ABS((_Axis.Axis.NcToPlc.ActTorque / 100) * ConfigChPeakCurrent);

		// Project slope from continuous stall torque/current
		ContStallCurrentEx := ContStallCurrent * 10.0;
		ContStallForceEx   := ContStallForce * 10.0;
		// Convert the actual current in amps to Nm
		IF CalculatedValues.ActCurrent = 0 THEN
			CalculatedValues.ActTorque := 0;
		ELSIF CalculatedValues.ActCurrent > 0 AND CalculatedValues.ActCurrent <= ContStallCurrentEx THEN
			IF ContStallCurrentEx > 0 THEN
				Scale					   := CalculatedValues.ActCurrent / ContStallCurrentEx;
				CalculatedValues.ActTorque := Scale * ContStallForceEx;
			END_IF
		END_IF

	1000: // Rotary or Linear Motor: Curve available - Compare actual torque value in Amps to the characteristic curve and output actual torque value in Nm
		CalculatedValues.ActCurrent := ABS((_Axis.Axis.NcToPlc.ActTorque / 100) * ConfigChPeakCurrent);
		// Convert the actual current in amps to Nm
		FOR i := 1 TO 9 DO
			IF CalculatedValues.ActCurrent = 0 THEN
				CalculatedValues.ActTorque := 0;
				EXIT;
			ELSIF CalculatedValues.ActCurrent > 0 AND CalculatedValues.ActCurrent < CalculatedValues.Curve.Iq[0] THEN
				IF CalculatedValues.Curve.Iq[0] > 0 THEN
					Scale					   := CalculatedValues.ActCurrent / CalculatedValues.Curve.Iq[0];
					CalculatedValues.ActTorque := Scale * CalculatedValues.Curve.M[0];
				END_IF

				EXIT;
			ELSIF CalculatedValues.ActCurrent >= CalculatedValues.Curve.Iq[i - 1] AND CalculatedValues.ActCurrent <= CalculatedValues.Curve.Iq[i] THEN
				IF (CalculatedValues.Curve.Iq[i] - CalculatedValues.Curve.Iq[i - 1]) > 0 AND CalculatedValues.ActCurrent - CalculatedValues.Curve.Iq[i - 1] > 0 THEN
					Scale					   := (CalculatedValues.ActCurrent - CalculatedValues.Curve.Iq[i - 1]) / (CalculatedValues.Curve.Iq[i] - CalculatedValues.Curve.Iq[i - 1]);
					CalculatedValues.ActTorque := (Scale * (CalculatedValues.Curve.M[i] - CalculatedValues.Curve.M[i - 1]) + CalculatedValues.Curve.M[i - 1]);
				END_IF

				EXIT;
			END_IF
		END_FOR

	5000: // Error state        
		SequenceState := -10;
END_CASE
END_METHOD

{attribute 'monitoring' := 'call'}
PROPERTY Error : BOOL
GET
Error := SequenceState = 5000;
END_GET
END_PROPERTY

{attribute 'monitoring' := 'call'}
PROPERTY ErrorId : UDINT
GET
ErrorId := _ErrorId;
END_GET
END_PROPERTY

